FUNCTION_BLOCK FB_SlaveArm
VAR
	//
	M_TESTfLAG:BOOL:=FALSE;
	m_jnt5Planner:Cubic_Polynomial_Interpolation;
	m_initAngle,m_initVel,m_initAcc,m_initT:REAL;
	m_targetAngle,m_targetVel,m_targetAcc:REAL;
	m_cmdAngle,m_cmdVel,m_cmdAcc:REAL;
	m_initFlag:BOOL:=FALSE;
	m_finishFlag:BOOL:=TRUE;
	m_endT:REAL:=5;
	m_dT:REAL:=0.0025;
	m_T:REAL:=0;
	// arm index, from 1 to 4
	m_armIdx: INT;
	
	// joints
	m_joints :ARRAY[1..g_sJntNum] OF FB_SlaveJoint;
	
	//  panel and insturment detect
	m_panelInstrumentOnIO AT%I*	:UDINT;
	m_panelDetect :FB_PanelDetect;
	m_instruDetect :FB_InstrumentDetect;
	m_instruNearDetect :FB_InstruNearDetect;
	m_panelOnFlag :BOOL:=FALSE;
	m_instruOnFlag :BOOL:=FALSE;
	m_instruNearFlag :BOOL:=FALSE;

	
	// trocar and  adjust detect
	m_adjustIO AT%I* :UDINT;
	m_adjustDetect :FB_AdjustDetect;
	m_trocarDetect : FB_TrocarDetect;
	m_adjustOnFlag :BOOL;
	m_trocarOnFlag :BOOL :=FALSE;
	m_adjustFallEdge :BOOL:=false;
	m_adjustFallEdgeDetect : F_TRIG;
	
	//arm light out to drive
	m_lightIO AT %Q* :DINT;
	
	//endoscope type and posture switch
	m_endoscopeTypeSwitch : FB_IOToggleCheck;
	m_endoscopePostureSwitch : FB_IOToggleCheck;
	
	// instrument instance
	m_instrument : FB_Instrument;
	
	// instrument invasion depth before it's unmounted
	m_instruInvasionDepth :LREAL;

	// arm cartesian data, defined in each arm origin
	m_curCartPose	:ST_Frame;
	m_curCartTwist: Vec6d;
	m_cmdCartTwist :Vec6d;
	m_cmdCartPose:ST_Frame;
	
	// arm joint data
	m_curMotorPos :Vec8d;
	m_curLinkPos :Vec8d;
	m_curLinkSingle :Vec8d;
	m_curJntPos :Vec8d;
	m_curDHJntPos :Vec6d;
	m_curGripAngle :LREAL;
	m_curJntVel :Vec8d;
	m_curDHJntVel :Vec6d;
	m_curJntTrq :Vec8d;
	m_rawJntCurrent :Vec8d;
	m_filtJntCurrent :Vec8d;
	m_cmdJntTrq :Vec8d;
	m_cmdJntCurrent : Vec8d;
	m_cmdJntPos :Vec8d;
	m_cmdJntVel :Vec8d;
		
	// arm dynamic data
	m_jntGravity : Vec8d:=g_zeroVec8d;
	m_jntMassMat : Mat3d;
	
	// arm jacobian and inverse
	m_jaco : Mat6d;
	
	// simulated status
	m_simJntPos :Vec8d;
	m_simDHJntPos :Vec6d;
	m_simGripAngle :LREAL;
	m_simCartPose : ST_Frame;
	m_simJaco : Mat6d;
	m_simJacoInv :Mat6d;
	m_isSingularity:BOOL:=false;
	
	// joint position controller
	m_jntPIDCtrl :ARRAY[1..g_sJntNum] OF FB_PID;
	
	// rising edge generator for instrument information reading
	m_ReadLDP:R_TRIG;
	
	// code execute time measure
	m_codeTime : Profiler;

	// output arm light
	m_SdoWrite:ARRAY [1..2] OF FB_EcCoESdoWrite;
	
	//IP of operating arm
	m_armNetId:T_AmsNetId; 	
	
	//Joint port number
	m_jointAddrJ8:UINT;	
	m_jointAddrPbox:UINT;	
	m_autoLogoutTon: TON;
	g_autoLogOutTRIG: R_TRIG;
	m_logStep: INT;
	m_actualNum: INT;
	m_registerNum: INT;
	m_register: INT;
	m_accountRepeat:BOOL;
	g_targetRatedCurrent: ARRAY[1..g_sJntNum] OF LREAL := [8(800)];

	
	fbSocketConnect      :FB_SocketConnect;
	fbSocketSend         :FB_SocketSend;;;
	fbSocketReceive      :FB_SocketReceive;
	bExecute:BOOL := TRUE;
	hSocket:T_hSocket;
	arrSendData: ARRAY [0..240] OF BYTE ;
	arrReadData: ARRAY [0..240] OF BYTE ;//read
	arrRFIDData: ARRAY [0..240] OF BYTE ;
	bSend   :BOOL;
	bReceive:BOOL;
	iStepRFID: INT;
	uiRFIDReadSN: ULINT;
	iStepRFIDOnLine: INT;
	fbTonRFID: TON;
	fbTonRFIDOnLine: TON;
	fbTonRFIDOnLineStep: TON;	
	g_offLineRFID:BOOL;
	m_offLineRFID:BOOL;
	
	fbTonCLK1:TON;
	fbTonCLK2:TON;
	
	uiRFIDRead:ULINT;
	wCRCReadSum:ULINT;
	g_readedRFID:BOOL;
	fbTonReadData:TON;
	
	
	wCRC16:WORD;
	g_moveMode:INT;
	g_energyType:INT;
	uiRFIDWrite:UINT;
	g_writedRFID:BOOL;
	
	g_RFIDinstruSN:ULINT;
	
	SNMid:INT;
	g_informationVerificationPassed:BOOL;
	g_instruSN:ULINT;
	m_writeRFIDTimes:DINT;
	m_writeInstrument_pos_L1:LREAL;
	m_writeInstrument_pos_L2:LREAL;
	m_writeInstrument_pos_L3:LREAL;
	m_readRFIDTimes:DINT;
	m_readInstrument_pos_L1:LREAL;
	m_readInstrument_pos_L2:LREAL;
	m_readInstrument_pos_L3:LREAL;
	
	fbTonRFIDReaded:TON;
	stateMachineMid: E_SlaveArmState;

	g_lastInstruJntPos: Vec5d;
	fbTon: TON;
	fbTon_Logout: TON;
	startFlag:BOOL;
	m_writeSdoStart: BOOL;
	m_writeSdoTimeStart: BOOL;
	m_writeSdoFinished: BOOL;
	m_SNWritten: BOOL;
	m_SNWriteStart: BOOL;
	m_bReadRecipeStep:   INT := 1;
	m_saveAccount:BOOL;
	m_saveCaliLinkEncoder:BOOL;
	RecipeManCommands:   RecipeManCommands;
	m_writePurposeSdoStart: BOOL;
	m_getSysTime:GETSYSTEMTIME;
	m_fileTime:T_FILETIME;
	m_time:STRING;
	m_timeNow:TIMESTRUCT;
	//mes
	m_serialNumOld:STRING;
	m_curTestCyclesOld:INT;
END_VAR

PROPERTY adjustFallEdge : BOOL
GET
adjustFallEdge := m_adjustFallEdge;
END_GET
END_PROPERTY

PROPERTY adjustOn : bool
GET
adjustOn := m_adjustOnFlag;
END_GET
END_PROPERTY

PROPERTY armIdx : int
GET
armIdx:=m_armIdx;
END_GET
END_PROPERTY

METHOD PROTECTED calcJaco : BOOL
VAR_IN_OUT CONSTANT
	i_DHJntPos :Vec6d;
END_VAR
VAR_IN_OUT
	r_jaco :Mat6d;
END_VAR
VAR_INPUT
END_VAR

VAR
	d1, L, a, b :LREAL;
	q3:LREAL;

	c1,c2,c4,c5,c6,c7 :LREAL;
	s1,s2,s4,s5,s6,s7 :LREAL;

END_VAR
d1:=GVL_SlaveArmKinematic.g_d1;
L:=m_instrument.instruTypeInfo.m_rodLength;
a:=m_instrument.instruTypeInfo.m_headLength;
b:=m_instrument.instruTypeInfo.m_fingerLength;

q3:=i_DHJntPos[3];
c1:=COS(i_DHJntPos[1]);
c2:=COS(i_DHJntPos[2]);
c4:=COS(i_DHJntPos[4]);
c5:=COS(i_DHJntPos[5]);
c6:=COS(i_DHJntPos[6]);

s1:=SIN(i_DHJntPos[1]);
s2:=SIN(i_DHJntPos[2]);
s4:=SIN(i_DHJntPos[4]);
s5:=SIN(i_DHJntPos[5]);
s6:=SIN(i_DHJntPos[6]);

// jacobian with DH joints
r_jaco[1,1]:=b*(c6*(c5*(c1*s4 - c2*c4*s1) + s1*s2*s5) - s6*(c1*c4 + c2*s1*s4)) + a*(c5*(c1*s4 - c2*c4*s1) + s1*s2*s5) - L*s1*s2 + q3*s1*s2;
r_jaco[1,2]:=-c1*(a*(c2*s5 + c4*c5*s2) - L*c2 + q3*c2 + b*(c6*(c2*s5 + c4*c5*s2) + s2*s4*s6));
r_jaco[1,3]:=-c1*s2;
r_jaco[1,4]:=s1*s2*(a*(c2*s5 + c4*c5*s2) + b*(c6*(c2*s5 + c4*c5*s2) + s2*s4*s6)) - c2*(b*(c6*(c5*(c1*s4 - c2*c4*s1) + s1*s2*s5) - s6*(c1*c4 + c2*s1*s4)) + a*(c5*(c1*s4 - c2*c4*s1) + s1*s2*s5));
r_jaco[1,5]:=- (a*(c2*s5 + c4*c5*s2) + b*(c6*(c2*s5 + c4*c5*s2) + s2*s4*s6))*(c1*c4 + c2*s1*s4) - s2*s4*(b*(c6*(c5*(c1*s4 - c2*c4*s1) + s1*s2*s5) - s6*(c1*c4 + c2*s1*s4)) + a*(c5*(c1*s4 - c2*c4*s1) + s1*s2*s5));
r_jaco[1,6]:= b*(c6*(c5*(c1*s4 - c2*c4*s1) + s1*s2*s5) - s6*(c1*c4 + c2*s1*s4))*(c2*c5 - c4*s2*s5) + b*(s5*(c1*s4 - c2*c4*s1) - c5*s1*s2)*(c6*(c2*s5 + c4*c5*s2) + s2*s4*s6);


r_jaco[2,1]:=0;
r_jaco[2,2]:=c1*(a*(c5*(s1*s4 + c1*c2*c4) - c1*s2*s5) + b*(c6*(c5*(s1*s4 + c1*c2*c4) - c1*s2*s5) - s6*(c4*s1 - c1*c2*s4)) + L*c1*s2 - q3*c1*s2) - s1*(b*(c6*(c5*(c1*s4 - c2*c4*s1) + s1*s2*s5) - s6*(c1*c4 + c2*s1*s4)) + a*(c5*(c1*s4 - c2*c4*s1) + s1*s2*s5) - L*s1*s2 + q3*s1*s2);
r_jaco[2,3]:= c2;
r_jaco[2,4]:=- s1*s2*(a*(c5*(s1*s4 + c1*c2*c4) - c1*s2*s5) + b*(c6*(c5*(s1*s4 + c1*c2*c4) - c1*s2*s5) - s6*(c4*s1 - c1*c2*s4))) - c1*s2*(b*(c6*(c5*(c1*s4 - c2*c4*s1) + s1*s2*s5) - s6*(c1*c4 + c2*s1*s4)) + a*(c5*(c1*s4 - c2*c4*s1) + s1*s2*s5));
r_jaco[2,5]:=(a*(c5*(s1*s4 + c1*c2*c4) - c1*s2*s5) + b*(c6*(c5*(s1*s4 + c1*c2*c4) - c1*s2*s5) - s6*(c4*s1 - c1*c2*s4)))*(c1*c4 + c2*s1*s4) - (b*(c6*(c5*(c1*s4 - c2*c4*s1) + s1*s2*s5) - s6*(c1*c4 + c2*s1*s4)) + a*(c5*(c1*s4 - c2*c4*s1) + s1*s2*s5))*(c4*s1 - c1*c2*s4);
r_jaco[2,6]:=b*(c6*(c5*(c1*s4 - c2*c4*s1) + s1*s2*s5) - s6*(c1*c4 + c2*s1*s4))*(s5*(s1*s4 + c1*c2*c4) + c1*c5*s2) - b*(s5*(c1*s4 - c2*c4*s1) - c5*s1*s2)*(c6*(c5*(s1*s4 + c1*c2*c4) - c1*s2*s5) - s6*(c4*s1 - c1*c2*s4));

r_jaco[3,1]:=a*(c5*(s1*s4 + c1*c2*c4) - c1*s2*s5) + b*(c6*(c5*(s1*s4 + c1*c2*c4) - c1*s2*s5) - s6*(c4*s1 - c1*c2*s4)) + L*c1*s2 - q3*c1*s2;
r_jaco[3,2]:=-s1*(a*(c2*s5 + c4*c5*s2) - L*c2 + q3*c2 + b*(c6*(c2*s5 + c4*c5*s2) + s2*s4*s6));
r_jaco[3,3]:=-s1*s2;
r_jaco[3,4]:=- c2*(a*(c5*(s1*s4 + c1*c2*c4) - c1*s2*s5) + b*(c6*(c5*(s1*s4 + c1*c2*c4) - c1*s2*s5) - s6*(c4*s1 - c1*c2*s4))) - c1*s2*(a*(c2*s5 + c4*c5*s2) + b*(c6*(c2*s5 + c4*c5*s2) + s2*s4*s6));
r_jaco[3,5]:=- (a*(c2*s5 + c4*c5*s2) + b*(c6*(c2*s5 + c4*c5*s2) + s2*s4*s6))*(c4*s1 - c1*c2*s4) - s2*s4*(a*(c5*(s1*s4 + c1*c2*c4) - c1*s2*s5) + b*(c6*(c5*(s1*s4 + c1*c2*c4) - c1*s2*s5) - s6*(c4*s1 - c1*c2*s4)));
r_jaco[3,6]:=b*(c6*(c5*(s1*s4 + c1*c2*c4) - c1*s2*s5) - s6*(c4*s1 - c1*c2*s4))*(c2*c5 - c4*s2*s5) + b*(c6*(c2*s5 + c4*c5*s2) + s2*s4*s6)*(s5*(s1*s4 + c1*c2*c4) + c1*c5*s2);

r_jaco[4,1]:=0;
r_jaco[4,2]:=-s1;
r_jaco[4,3]:=0;
r_jaco[4,4]:=-c1*s2;
r_jaco[4,5]:=c1*c2*s4 - c4*s1;
r_jaco[4,6]:=s5*(s1*s4 + c1*c2*c4) + c1*c5*s2;

r_jaco[5,1]:=-1;
r_jaco[5,2]:=0;
r_jaco[5,3]:=0;
r_jaco[5,4]:=c2;
r_jaco[5,5]:=s2*s4;
r_jaco[5,6]:=c4*s2*s5 - c2*c5;

r_jaco[6,1]:=0;
r_jaco[6,2]:=c1;
r_jaco[6,3]:=0;
r_jaco[6,4]:=-s1*s2;
r_jaco[6,5]:=c1*c4 + c2*s1*s4;
r_jaco[6,6]:=c5*s1*s2 - s5*(c1*s4 - c2*c4*s1);
END_METHOD

METHOD PROTECTED checkIO : BOOL

VAR

	i: INT;
	ReturnDwordRead:DWORD;
	ReturnDwordWrite:DWORD;
END_VAR
// check adjust button
m_adjustOnFlag := m_adjustDetect.run(m_adjustIO);
m_adjustFallEdgeDetect(CLK:=m_adjustOnFlag, Q=>m_adjustFallEdge);

// check trocar
m_trocarOnFlag := m_trocarDetect.run(m_adjustIO);

// check panel and instrument
m_panelOnFlag := m_panelDetect.run(m_panelInstrumentOnIO);
m_instruOnFlag :=m_instruDetect.run(m_panelInstrumentOnIO);
m_instruNearFlag := m_instruNearDetect.run(m_panelInstrumentOnIO);

//read instrument information
IF FALSE = m_instruOnFlag THEN
	m_instrument.reset();
END_IF


m_ReadLDP(CLK:= m_instruOnFlag, Q=>startFlag );
// try to read again if instrument ID is undefined
startFlag := startFlag OR m_instrument.onChipData.m_ErrorID = 1 OR GVL_InstruTestUIVars.g_readInstruinformation;
m_instrument.readParameters(startFlag);

GVL_InstruTestUIVars.g_readInstruinformationFlag:=m_instrument.onChipData.m_InstruReadSucceed;
// check endoscope type and posture 
IF m_endoscopeTypeSwitch.check((m_panelInstrumentOnIO AND 16#20)=32) THEN
	IF m_instrument.curScopeType = EndoScopeType_30 THEN
		m_instrument.nextScopeType := EndoscopeType_0;
	ELSE
		m_instrument.nextScopeType := EndoscopeType_30;
	END_IF
END_IF
IF m_endoscopePostureSwitch.check((m_panelInstrumentOnIO AND 16#10)=16) AND m_instrument.curScopeType = EndoScopeType_30  THEN
	IF m_instrument.curScopePosture = EndoScopePosture_HeadDown THEN
		m_instrument.nextScopePosture := EndoscopePosture_HeadUp;
	ELSE
		m_instrument.nextScopePosture := EndoScopePosture_HeadDown;
	END_IF
END_IF

IF GVL_InstruTestUIVars.g_incInstruNumOfUses THEN
	GVL_InstruTestUIVars.g_jnt5RotateFlag:=TRUE;
	m_writeSdoTimeStart := TRUE;
ELSE
	IF m_writeSdoTimeStart THEN
		IF   NOT m_writeSdoFinished THEN
			m_writeSdoFinished :=instrument.addNumOfUseToChip();

		ELSE
			m_writeSdoTimeStart :=FALSE;
			m_writeSdoFinished:=FALSE;
		END_IF
	END_IF
END_IF

IF GVL_InstruTestUIVars.g_clearInstruNumOfUses THEN
	m_writeSdoStart := TRUE;
ELSE
	IF m_writeSdoStart THEN
		IF   NOT m_writeSdoFinished THEN
			m_writeSdoFinished :=instrument.clearNumOfUseToChip();

		ELSE
			m_writeSdoStart :=FALSE;
			m_writeSdoFinished:=FALSE;
		END_IF
	END_IF
END_IF

// write SN to CoE
IF GVL_InstruTestUIVars.g_writeSNFlag THEN
	m_SNWriteStart := TRUE;
ELSE
	IF m_SNWriteStart THEN
		IF   NOT m_SNWritten THEN
			m_SNWritten := instrument.writeSNToChip(STRING_TO_ULINT(GVL_InstruTestUIVars.g_newInstruSN));
		ELSE
			m_SNWriteStart :=FALSE;
			m_SNWritten:=FALSE;
		END_IF
	END_IF
END_IF

IF GVL_InstruTestUIVars.g_writeInstruPurpose AND m_instrument.onChipData.m_InstruReadSucceed THEN
	m_writePurposeSdoStart := TRUE;
ELSE
	IF m_writePurposeSdoStart THEN
		IF   NOT m_writeSdoFinished THEN
			m_writeSdoFinished :=instrument.writePurpose();

		ELSE
			m_writePurposeSdoStart :=FALSE;
			m_writeSdoFinished:=FALSE;
		END_IF
	END_IF
END_IF

GVL_InstruTestUIVars.g_maxAngle:=INT_TO_REAL(REAL_TO_INT(m_instrument.instruTypeInfo.m_maxGripAngle/g_deg2Rad));
GVL_InstruTestUIVars.g_maxRoll:=INT_TO_REAL(REAL_TO_INT(m_instrument.instruTypeInfo.m_rollLimit/g_deg2Rad));
GVL_InstruTestUIVars.g_maxPitch:=INT_TO_REAL(REAL_TO_INT(m_instrument.instruTypeInfo.m_pitchLimit/g_deg2Rad));
GVL_InstruTestUIVars.g_maxYaw:=INT_TO_REAL(REAL_TO_INT(m_instrument.instruTypeInfo.m_yawLimit/g_deg2Rad));
GVL_InstruTestUIVars.g_maxAngleEnable:=GVL_InstruTestUIVars.g_targetGripAng*g_deg2rad>m_instrument.instruTypeInfo.m_maxGripAngle;
GVL_InstruTestUIVars.g_maxRollEnable:=ABS(GVL_InstruTestUIVars.g_targetRollAng)*g_deg2rad>m_instrument.instruTypeInfo.m_rollLimit;
GVL_InstruTestUIVars.g_maxPitchEnable:=ABS(GVL_InstruTestUIVars.g_targetPitchAng)*g_deg2rad>m_instrument.instruTypeInfo.m_pitchLimit;
GVL_InstruTestUIVars.g_maxYawEnable:=ABS(GVL_InstruTestUIVars.g_targetYawAng)*g_deg2rad>m_instrument.instruTypeInfo.m_yawLimit;

GVL_InstruTestUIVars.g_incInstruNumOfUses:=FALSE;
GVL_InstruTestUIVars.g_clearInstruNumOfUses:=FALSE;
GVL_InstruTestUIVars.g_writeSNFlag:=FALSE;
GVL_InstruTestUIVars.g_writeInstruPurpose:=FALSE;

GVL_InstruTestUIVars.g_instruNumberOfUses:=ULINT_TO_UINT( m_instrument.onChipData.m_InstruusageCounts);
GVL_InstruTestUIVars.g_instruNumberOfAllUses:=ULINT_TO_UINT( m_instrument.onChipData.m_InstruUsageCounts);
GVL_InstruTestUIVars.g_readInstruPurpose:=ULINT_TO_UINT( m_instrument.onChipData.m_InstruPurpose);
GVL_InstruTestUIVars.g_readPurposeTime:=ULINT_TO_UINT( m_instrument.onChipData.m_InstruPurposeTime);

GVL_InstruTestUIVars.g_instruSN:=ULINT_TO_STRING(m_instrument.onChipData.m_InstruseriesNum);
IF (LEN(GVL_InstruTestUIVars.g_instruSN)=10)THEN
	GVL_InstruTestUIVars.g_instruSN:=concat('00',GVL_InstruTestUIVars.g_instruSN);
ELSIF  (LEN(GVL_InstruTestUIVars.g_instruSN)=11)THEN
	GVL_InstruTestUIVars.g_instruSN:=concat('0',GVL_InstruTestUIVars.g_instruSN);
ELSE
	GVL_InstruTestUIVars.g_instruSN:=GVL_InstruTestUIVars.g_instruSN;
END_IF

GVL_InstruTestUIVars.g_rotationActualCurrent:=m_filtJntCurrent[7];
GVL_InstruTestUIVars.g_pitchActualCurrent:=m_filtJntCurrent[6];
GVL_InstruTestUIVars.g_deviationActualCurrent:=m_filtJntCurrent[4];
//***************************修改电流极限**************************//
GVL_InstruTestUIVars.g_actualRatedCurrent:=g_targetRatedCurrent;
IF GVL_InstruTestUIVars.g_modifyRatedCurrent THEN
	GVL_InstruTestUIVars.g_modifyRatedCurrent:=FALSE;
	FOR i:=1 TO 8 BY 1 DO 
		GVL_InstruTestUIVars.g_actualRatedCurrent[i]:=GVL_InstruTestUIVars.g_targetRatedCurrent;
		g_targetRatedCurrent[i]:=GVL_InstruTestUIVars.g_targetRatedCurrent;
	END_FOR
END_IF
IF GVL_InstruTestUIVars.g_rotationTargetCurrent=0 THEN GVL_InstruTestUIVars.g_rotationTargetCurrent:=100; END_IF
IF GVL_InstruTestUIVars.g_pitchTargetCurrent=0 THEN GVL_InstruTestUIVars.g_pitchTargetCurrent:=100; END_IF
IF GVL_InstruTestUIVars.g_deviationTargetCurrent=0 THEN GVL_InstruTestUIVars.g_deviationTargetCurrent:=100; END_IF
IF GVL_InstruTestUIVars.g_deviationTargetCurrent=0 THEN GVL_InstruTestUIVars.g_deviationTargetCurrent:=100; END_IF
IF GVL_InstruTestUIVars.g_account.actualPermission=2 AND GVL_InstruTestUIVars.g_stateMachine=SlaveArmState_InstruManualTest  THEN
	GVL_InstruTestUIVars.g_actualRatedCurrent[7]:=GVL_InstruTestUIVars.g_rotationTargetCurrent;
	GVL_InstruTestUIVars.g_actualRatedCurrent[6]:=GVL_InstruTestUIVars.g_pitchTargetCurrent;
	GVL_InstruTestUIVars.g_actualRatedCurrent[5]:=GVL_InstruTestUIVars.g_deviationTargetCurrent;
	GVL_InstruTestUIVars.g_actualRatedCurrent[4]:=GVL_InstruTestUIVars.g_deviationTargetCurrent;
END_IF
IF GVL_InstruTestUIVars.g_stateMachine=SlaveArmState_InstruAutoTest AND GVL_MES.g_autoTestMode=3 THEN
	GVL_InstruTestUIVars.g_actualRatedCurrent[4]:=540;
	GVL_InstruTestUIVars.g_actualRatedCurrent[5]:=540;
	GVL_InstruTestUIVars.g_actualRatedCurrent[6]:=540;
	GVL_InstruTestUIVars.g_actualRatedCurrent[7]:=540;
	IF m_instrument.onChipData.m_InstruReadSucceed AND(InstruType_CauteryHook=m_instrument.m_instruType OR InstruType_CauterySpatula=m_instrument.m_instruType) THEN
	GVL_InstruTestUIVars.g_actualRatedCurrent[4]:=270;
	GVL_InstruTestUIVars.g_actualRatedCurrent[5]:=270;
	GVL_InstruTestUIVars.g_actualRatedCurrent[6]:=270;
	GVL_InstruTestUIVars.g_actualRatedCurrent[7]:=270;
	END_IF
END_IF
//Account
GVL_InstruTestUIVars.g_account.memoryAccountNumber[0] :='admin';
GVL_InstruTestUIVars.g_account.memoryPassWord[0] :='yfAGIBOT2025';
GVL_InstruTestUIVars.g_account.memoryPermission[0] :=1;
GVL_InstruTestUIVars.g_account.memoryName[0] :='admin';
GVL_InstruTestUIVars.g_account.memoryWorkNum[0] :=101;
GVL_InstruTestUIVars.g_account.memoryDisable[0]:=FALSE;
CASE m_logStep OF 
	0: 
	  IF GVL_InstruTestUIVars.g_account.logOn THEN 
		   m_logStep:=5;
		   m_actualNum:=-1;
		  GVL_InstruTestUIVars.g_account.logOn:=FALSE;
	  END_IF
	5:
	FOR i:= 0 TO 50 BY 1 DO
		IF GVL_InstruTestUIVars.g_account.actualAccountNumber = GVL_InstruTestUIVars.g_account.memoryAccountNumber[i] AND GVL_InstruTestUIVars.g_account.actualAccountNumber <> ''THEN
			m_actualNum:=i;
			m_logStep:=10;
		ELSE
			IF m_actualNum=-1 THEN
				GVL_InstruTestUIVars.g_account.prompt:='Account Err';
				m_logStep:=0;
			END_IF
		END_IF
	END_FOR
	10:
	IF GVL_InstruTestUIVars.g_account.actualPassWord = GVL_InstruTestUIVars.g_account.memoryPassWord[m_actualNum] AND GVL_InstruTestUIVars.g_account.actualAccountNumber <> ''THEN
		m_logStep:=12;
	ELSE
		GVL_InstruTestUIVars.g_account.prompt:='PassWord Err';
		m_logStep:=0;
	END_IF
	12:
	IF GVL_InstruTestUIVars.g_account.memoryDisable[m_actualNum] THEN
		GVL_InstruTestUIVars.g_account.prompt:='No Enable';
		m_logStep:=0;
	ELSE
		m_logStep:=15;
	END_IF
	15:
	GVL_InstruTestUIVars.g_account.actualPermission := GVL_InstruTestUIVars.g_account.memoryPermission[m_actualNum];
	GVL_InstruTestUIVars.g_account.actualWorkNum := GVL_InstruTestUIVars.g_account.memoryWorkNum[m_actualNum];
	GVL_InstruTestUIVars.g_account.actualName := GVL_InstruTestUIVars.g_account.memoryName[m_actualNum];
	GVL_InstruTestUIVars.g_account.autoLogOut:=FALSE;
	GVL_InstruTestUIVars.g_account.prompt:='Login Succeeded';
	m_logStep:=0;
END_CASE

FOR i:=1 TO 5 DO 
	IF stateMachineMid<>GVL_InstruTestUIVars.g_stateMachine OR ABS(GVL_InstruTestUIVars.g_curInstruJntPos[i]-g_lastInstruJntPos[i])>0.01 THEN
		GVL_InstruTestUIVars.g_account.autoLogOut:=FALSE;
	ELSE
		IF NOT GVL_InstruTestUIVars.g_account.autoLogOut THEN 
			IF fbTon_Logout.Q THEN
				GVL_InstruTestUIVars.g_account.autoLogOut:=TRUE;
			END_IF
		END_IF
	END_IF
END_FOR
	fbTon(IN:= NOT fbTon.Q, PT:=T#10MS );
	IF fbTon.Q THEN
		g_lastInstruJntPos:= GVL_InstruTestUIVars.g_curInstruJntPos;
	END_IF
stateMachineMid:=GVL_InstruTestUIVars.g_stateMachine;
fbTon_Logout(IN:=NOT GVL_InstruTestUIVars.g_account.autoLogOut,PT:=T#0.1S);


m_autoLogoutTon(IN:=GVL_InstruTestUIVars.g_account.autoLogOut,PT:=T#1H);
g_autoLogOutTRIG(CLK:=m_autoLogoutTon.Q);
IF GVL_InstruTestUIVars.g_account.logOut OR g_autoLogOutTRIG.Q THEN
	GVL_InstruTestUIVars.g_account.actualPermission :=0;
	GVL_InstruTestUIVars.g_account.actualAccountNumber :='';
	GVL_InstruTestUIVars.g_account.actualPassWord :='';
	GVL_InstruTestUIVars.g_account.actualWorkNum :=0;
	GVL_InstruTestUIVars.g_account.actualName :='';
	GVL_InstruTestUIVars.g_account.logOut:=FALSE;
	GVL_InstruTestUIVars.g_account.prompt:='';
END_IF
IF GVL_InstruTestUIVars.g_clearInformation THEN
	GVL_InstruTestUIVars.g_account.actualAccountNumber :='';
	GVL_InstruTestUIVars.g_account.actualPassWord :='';
	GVL_InstruTestUIVars.g_account.actualWorkNum :=0;
	GVL_InstruTestUIVars.g_account.actualName :='';
	GVL_InstruTestUIVars.g_account.prompt:='';
	GVL_InstruTestUIVars.g_account.registerAccountNumber :='';
	GVL_InstruTestUIVars.g_account.registerPassWord :='';
	GVL_InstruTestUIVars.g_account.registerWorkNum :=0;
	GVL_InstruTestUIVars.g_account.registerName :='';
	GVL_InstruTestUIVars.g_account.prompt:='';
	GVL_InstruTestUIVars.g_clearInformation:=FALSE;
END_IF
IF GVL_InstruTestUIVars.g_account.registerPermission<>2 AND GVL_InstruTestUIVars.g_account.registerPermission<>3 AND
	GVL_InstruTestUIVars.g_account.registerPermission<>4 THEN
//	GVL_InstruTestUIVars.g_account.registerPermission:=4;
END_IF
m_getSysTime(timeLoDW=>m_fileTime.dwLowDateTime, timeHiDW=>m_fileTime.dwHighDateTime);
m_timeNow:=FILETIME_TO_SYSTEMTIME(m_fileTime);
m_timeNow.wHour:=m_timeNow.wHour+8;
IF m_timeNow.wHour>23 THEN
	m_timeNow.wHour:=m_timeNow.wHour-24;
END_IF
m_time:=SYSTEMTIME_TO_STRING(m_timeNow);
CASE m_registerNum OF 
	0:
	  IF GVL_InstruTestUIVars.g_account.register THEN 
		  GVL_InstruTestUIVars.g_account.register:=FALSE;
		  GVL_InstruTestUIVars.g_account.prompt:='';
		  m_accountRepeat:=FALSE;
		  m_register:=-1;
		  m_registerNum:=5;
	  END_IF
	5:
	FOR i:= 0 TO 50 BY 1 DO
      IF  GVL_InstruTestUIVars.g_account.registerAccountNumber <> GVL_InstruTestUIVars.g_account.memoryAccountNumber[i] AND GVL_InstruTestUIVars.g_account.registerAccountNumber <> ''THEN
		;	  
	  ELSE
		  m_accountRepeat:=TRUE;
	  END_IF
	END_FOR
	m_registerNum:=6;
	6:
	IF m_accountRepeat THEN
		GVL_InstruTestUIVars.g_account.prompt:='Account Repeat';
		m_registerNum:=0;
	ELSE
		m_registerNum:=10;
	END_IF
	10:
	IF GVL_InstruTestUIVars.g_account.registerPassWord<> '' THEN
		m_registerNum:=15;
	ELSE
		GVL_InstruTestUIVars.g_account.prompt:='No PassWord';
		m_registerNum:=0;
	END_IF
	15:
	IF GVL_InstruTestUIVars.g_account.registerWorkNum<> 0 THEN
		m_registerNum:=20;
	ELSE
		GVL_InstruTestUIVars.g_account.prompt:='No WorkNum';
		m_registerNum:=0;
	END_IF
	20:
	IF GVL_InstruTestUIVars.g_account.registerName<> '' THEN
		m_registerNum:=25;
	ELSE
		GVL_InstruTestUIVars.g_account.prompt:='No Name';
		m_registerNum:=0;
	END_IF
	25:
	IF GVL_InstruTestUIVars.g_account.registerPermission<> 0 THEN
		m_registerNum:=30;
	ELSE
		GVL_InstruTestUIVars.g_account.prompt:='No Permission';
		m_registerNum:=0;
	END_IF
	30:
	FOR i:= 50 TO 0 BY -1 DO
      IF  '' = GVL_InstruTestUIVars.g_account.memoryAccountNumber[i] THEN
		 m_register:=i;
		 m_registerNum:=35;
	  ELSE
		  IF m_register=-1 THEN
			 GVL_InstruTestUIVars.g_account.prompt:='No Room';
			 m_registerNum:=0;	
		END_IF
	  END_IF
 	END_FOR
	35:
	GVL_InstruTestUIVars.g_account.memoryAccountNumber[m_register]:=GVL_InstruTestUIVars.g_account.registerAccountNumber;
	GVL_InstruTestUIVars.g_account.memoryPassWord[m_register]:=GVL_InstruTestUIVars.g_account.registerPassWord;
	GVL_InstruTestUIVars.g_account.memoryWorkNum[m_register]:=GVL_InstruTestUIVars.g_account.registerWorkNum;
	GVL_InstruTestUIVars.g_account.memoryName[m_register]:=GVL_InstruTestUIVars.g_account.registerName;
	GVL_InstruTestUIVars.g_account.memoryPermission[m_register]:=GVL_InstruTestUIVars.g_account.registerPermission;
	IF GVL_InstruTestUIVars.g_account.registerPermission=1 THEN
		GVL_InstruTestUIVars.g_account.memoryPermission[m_register]:=4;
	END_IF
	GVL_InstruTestUIVars.g_account.memoryTime[m_register]:=m_time;
	GVL_InstruTestUIVars.g_account.prompt:='Register Succeeded';
	m_registerNum:=0;
	m_saveAccount:=TRUE;
END_CASE

GVL_InstruTestUIVars.g_accountSN := LIMIT(1,GVL_InstruTestUIVars.g_accountSN, 50);
IF GVL_InstruTestUIVars.g_accountDelete THEN 
	GVL_InstruTestUIVars.g_accountDelete:=FALSE;
	m_saveAccount:=TRUE;
	GVL_InstruTestUIVars.g_account.memoryAccountNumber[GVL_InstruTestUIVars.g_accountSN]:='';
	GVL_InstruTestUIVars.g_account.memoryPassWord[GVL_InstruTestUIVars.g_accountSN]:='';
	GVL_InstruTestUIVars.g_account.memoryWorkNum[GVL_InstruTestUIVars.g_accountSN]:=0;
	GVL_InstruTestUIVars.g_account.memoryName[GVL_InstruTestUIVars.g_accountSN]:='';
	GVL_InstruTestUIVars.g_account.memoryPermission[GVL_InstruTestUIVars.g_accountSN]:=0;
	GVL_InstruTestUIVars.g_account.memoryTime[GVL_InstruTestUIVars.g_accountSN]:='';
END_IF
IF GVL_InstruTestUIVars.g_disableAccount THEN 
	GVL_InstruTestUIVars.g_disableAccount:=FALSE;
	IF GVL_InstruTestUIVars.g_account.memoryDisable[GVL_InstruTestUIVars.g_accountSN] THEN
		GVL_InstruTestUIVars.g_account.memoryDisable[GVL_InstruTestUIVars.g_accountSN]:=FALSE;
	ELSE
		GVL_InstruTestUIVars.g_account.memoryDisable[GVL_InstruTestUIVars.g_accountSN]:=TRUE;
	END_IF
END_IF	
FOR i:=1 TO 50 BY 1 DO 
	IF GVL_InstruTestUIVars.g_account.memoryAccountNumber[i]='' THEN
		GVL_InstruTestUIVars.g_account.memoryDisable[i]:=FALSE;
	END_IF
END_FOR
GVL_InstruTestUIVars.g_queryAccountSN := LIMIT(0,GVL_InstruTestUIVars.g_queryAccountSN, 50);
IF GVL_InstruTestUIVars.g_queryAccountFlag THEN 
	GVL_InstruTestUIVars.g_queryAccountFlag:=FALSE;
	GVL_InstruTestUIVars.g_queryAccountNumber:='';
	GVL_InstruTestUIVars.g_queryPassWord:='';
	GVL_InstruTestUIVars.g_queryPermission:=0;
	GVL_InstruTestUIVars.g_queryWorkNum:=0;
	GVL_InstruTestUIVars.g_queryName:='';
	GVL_InstruTestUIVars.g_queryTime:='';
	GVL_InstruTestUIVars.g_queryAccountNumber:=GVL_InstruTestUIVars.g_account.memoryAccountNumber[GVL_InstruTestUIVars.g_queryAccountSN];
	GVL_InstruTestUIVars.g_queryPassWord:=GVL_InstruTestUIVars.g_account.memoryPassWord[GVL_InstruTestUIVars.g_queryAccountSN];
	GVL_InstruTestUIVars.g_queryPermission:=GVL_InstruTestUIVars.g_account.memoryPermission[GVL_InstruTestUIVars.g_queryAccountSN];
	GVL_InstruTestUIVars.g_queryWorkNum:=GVL_InstruTestUIVars.g_account.memoryWorkNum[GVL_InstruTestUIVars.g_queryAccountSN];
	GVL_InstruTestUIVars.g_queryName:=GVL_InstruTestUIVars.g_account.memoryName[GVL_InstruTestUIVars.g_queryAccountSN];
	GVL_InstruTestUIVars.g_queryTime:=GVL_InstruTestUIVars.g_account.memoryTime[GVL_InstruTestUIVars.g_queryAccountSN];
END_IF
IF GVL_InstruTestUIVars.g_queryClear THEN 
	GVL_InstruTestUIVars.g_queryClear:=FALSE;
	GVL_InstruTestUIVars.g_queryAccountNumber:='';
	GVL_InstruTestUIVars.g_queryPassWord:='';
	GVL_InstruTestUIVars.g_queryPermission:=0;
	GVL_InstruTestUIVars.g_queryWorkNum:=0;
	GVL_InstruTestUIVars.g_queryName:='';
	GVL_InstruTestUIVars.g_queryTime:='';
END_IF

bExecute:=NOT fbSocketConnect.bError OR fbTon.Q;

fbSocketConnect(
	sSrvNetId:= , 
	sRemoteHost:='192.168.1.202' , 
	nRemotePort:= 4196, 
	bExecute:= bExecute, 
	tTimeout:=T#3S , 
	bBusy=> , 
	bError=> , 
	nErrId=> , 
	hSocket=>hSocket );
	
	fbSocketSend(
	sSrvNetId:= , 
	hSocket:= hSocket, 
	cbLen:= SIZEOF(arrSendData), 
	pSrc:= ADR(arrSendData), 
	bExecute:= bSend, 
	tTimeout:= T#3S, 
	bBusy=> , 
	bError=> , 
	nErrId=> );
	
	
	fbSocketReceive(
	sSrvNetId:= , 
	hSocket:=hSocket , 
	cbLen:= SIZEOF(arrReadData), 
	pDest:= ADR(arrReadData), 
	bExecute:= bReceive, 
	tTimeout:= T#3S, 
	bBusy=> , 
	bError=> , 
	nErrId=> , 
	nRecBytes=> );
	
	bSend:=FALSE;
	fbTonCLK1(IN:=NOT fbTonCLK2.Q,PT:=T#1S);
	fbTonCLK2(IN:=fbTonCLK1.Q,PT:=T#1S);
	bReceive:=fbTonCLK1.Q;
//RFID
m_instrument.readParametersRFID(GVL_InstruTestUIVars.g_readRFID);
GVL_InstruTestUIVars.g_readRFID:=FALSE;
g_informationVerificationPassed:=FALSE;
IF m_instrument.onChipData.m_InstruReadSucceedRFID AND m_instrument.onChipData.m_InstruseriesNumRFID=m_instrument.onChipData.m_InstruseriesNum  AND 
	ABS(m_instrument.onChipData.m_InstruPosRFID[1]-m_instrument.onChipData.m_InstruPos[1])<0.01 AND
	ABS(m_instrument.onChipData.m_InstruPosRFID[2]-m_instrument.onChipData.m_InstruPos[2])<0.01 AND
	ABS(m_instrument.onChipData.m_InstruPosRFID[3]-m_instrument.onChipData.m_InstruPos[3])<0.01 THEN
	
	g_informationVerificationPassed:=TRUE;
END_IF;
GVL_InstruTestUIVars.g_RFID_SN:=ULINT_TO_STRING(m_instrument.onChipData.m_InstruseriesNumRFID);
IF (LEN(GVL_InstruTestUIVars.g_RFID_SN)=10)THEN
	GVL_InstruTestUIVars.g_RFID_SN:=concat('00',GVL_InstruTestUIVars.g_RFID_SN);
ELSIF  (LEN(GVL_InstruTestUIVars.g_RFID_SN)=11)THEN
	GVL_InstruTestUIVars.g_RFID_SN:=concat('0',GVL_InstruTestUIVars.g_RFID_SN);
ELSE
	GVL_InstruTestUIVars.g_RFID_SN:=GVL_InstruTestUIVars.g_RFID_SN;
END_IF
GVL_InstruTestUIVars.m_RFIDTimes:=ULINT_TO_DINT(m_instrument.onChipData.m_InstruUsageCountsRFID);
GVL_InstruTestUIVars.m_Instrument_pos_L1:=m_instrument.onChipData.m_InstruPosRFID[1];
GVL_InstruTestUIVars.m_Instrument_pos_L2:=m_instrument.onChipData.m_InstruPosRFID[2];
GVL_InstruTestUIVars.m_Instrument_pos_L3:=m_instrument.onChipData.m_InstruPosRFID[3];
GVL_InstruTestUIVars.g_informationVerificationPassed:=g_informationVerificationPassed;
GVL_InstruTestUIVars.g_readedRFID:=m_instrument.onChipData.m_InstruReadSucceedRFID;
IF GVL_InstruTestUIVars.g_readRFID AND iStepRFID=0 THEN
	GVL_InstruTestUIVars.g_readRFID:=FALSE;
	g_readedRFID:=FALSE;
	GVL_InstruTestUIVars.g_readRFIDFlag:=FALSE;
	uiRFIDReadSN:=0;
	iStepRFID:=3;
	iStepRFIDOnLine:=0;
END_IF
IF GVL_InstruTestUIVars.g_writeRFID AND iStepRFID=0 THEN
	GVL_InstruTestUIVars.g_writeRFID:=FALSE;
	iStepRFID:=53;
	iStepRFIDOnLine:=0;
END_IF

fbTonRFID(IN:=iStepRFID=10 OR iStepRFID=60, PT:=T#5S , Q=> , ET=> );
fbTonRFIDOnLine(IN:=m_offLineRFID , PT:=T#2S , Q=> , ET=> );
fbTonRFIDOnLineStep(IN:=iStepRFIDOnLine=10 , PT:=T#1S , Q=> , ET=> );
fbTonReadData(IN:=iStepRFID=15 OR iStepRFID=65 , PT:=T#0.5S , Q=> , ET=> );
IF fbTonRFIDOnLine.Q THEN
    g_offLineRFID:=FALSE;;
END_IF

CASE iStepRFID OF
	0:
(*		CASE iStepRFIDOnLine OF   //On  Off line
			0:
			  arrReadData:=arrRFIDData;
			  arrSendData:=arrRFIDData;
			  iStepRFIDOnLine:=5;
			5:   
			  arrSendData[1]:=16#FF;
			  arrSendData[2]:=16#08;  arrSendData[3]:=16#11;
			  arrSendData[4]:=16#00;  arrSendData[5]:=16#01;
			  arrSendData[6]:=16#00;  arrSendData[7]:=16#00;
			  arrSendData[8]:=16#01;  arrSendData[9]:=16#EF;
			  arrSendData[10]:=16#7F;  arrSendData[11]:=16#32;
			  bSend:=TRUE; 
			  iStepRFIDOnLine:=10;
			10:
			  IF arrReadData[0]<>0  THEN
				  g_offLineRFID:=TRUE;
				  m_offLineRFID:=FALSE;
			  ELSE
                  m_offLineRFID:=TRUE;
			  END_IF
			  IF fbTonRFIDOnLineStep.Q THEN
			  	  iStepRFIDOnLine:=0;
			  END_IF
		END_CASE
		
	*)	
    3:                           //Read
	  arrReadData:=arrRFIDData;
	  arrSendData:=arrRFIDData;
	  iStepRFID:=5;
	5:
	  arrSendData[0]:=16#FF;
	  arrSendData[1]:=16#08;  arrSendData[2]:=16#11;
	  arrSendData[3]:=16#00;  arrSendData[4]:=16#01;
	  arrSendData[5]:=16#00;  arrSendData[6]:=16#00;
	  arrSendData[7]:=16#01;  arrSendData[8]:=16#6E;
	  arrSendData[9]:=16#1F;  arrSendData[10]:=16#F2;
	  arrSendData[11]:=16#00; 
	  bSend:=TRUE; 
	  iStepRFID:=10;
	10:
	   IF arrReadData[0]<>0  THEN
		   iStepRFID:=15;
	   END_IF
	   IF fbTonRFID.Q THEN
		   iStepRFID:=0;
	       iStepRFIDOnLine:=0;
	   END_IF
	15: 
	IF fbTonReadData.Q THEN
//	   IF arrReadData[5]=0 THEN
	   	   iStepRFID:=20;
//	   END_IF
//	   IF arrReadData[5]<>0THEN
//	   	   iStepRFID:=30;
//	   END_IF
	END_IF
    20:
	   uiRFIDRead:=0;
	   FOR i:=8 TO 108 BY 1 DO
		    uiRFIDRead:=BYTE_TO_UINT(arrReadData[i])+uiRFIDRead;
	   END_FOR
  	   iStepRFID:=25;
	 25:
//	   AryByteTo(In:=arrReadData[111] , Size:= 2, Order:=_eBYTE_ORDER._HIGH_LOW , OutVal:=wCRCReadSum );
	   wCRCReadSum:=SHL(BYTE_TO_ULINT(arrReadData[109]),8)OR BYTE_TO_ULINT(arrReadData[110]);
	   IF wCRCReadSum=uiRFIDRead THEN
	    	g_readedRFID:=TRUE;
			GVL_InstruTestUIVars.g_readRFIDFlag:=TRUE;
			uiRFIDReadSN:=0;
	   FOR i:=1 TO 8 BY 1 DO
		  uiRFIDReadSN:=SHL(BYTE_TO_ULINT(arrReadData[58+i]),64-i*8)+uiRFIDReadSN;
	  END_FOR
	  m_readRFIDTimes:=0;
	   FOR i:=1 TO 4 BY 1 DO
		  m_readRFIDTimes:=SHL(BYTE_TO_DINT(arrReadData[68+i]),32-i*8)+m_readRFIDTimes;
	  END_FOR
	  m_readInstrument_pos_L1:=0;
	  m_readInstrument_pos_L2:=0;
	  m_readInstrument_pos_L3:=0;
	   FOR i:=1 TO 4 BY 1 DO
		  m_readInstrument_pos_L1:=DINT_TO_LREAL(SHL(BYTE_TO_DINT(arrReadData[28+i]),32-i*8))/1000+m_readInstrument_pos_L1;
	  END_FOR
	   FOR i:=1 TO 4 BY 1 DO
		  m_readInstrument_pos_L2:=DINT_TO_LREAL(SHL(BYTE_TO_DINT(arrReadData[38+i]),32-i*8))/1000+m_readInstrument_pos_L2;
	  END_FOR
	   FOR i:=1 TO 4 BY 1 DO
		  m_readInstrument_pos_L3:=DINT_TO_LREAL(SHL(BYTE_TO_DINT(arrReadData[48+i]),32-i*8))/1000+m_readInstrument_pos_L3;
	  END_FOR
	  
//			AryByteTo(In:=arrReadData[61] , Size:= 12, Order:=_eBYTE_ORDER._HIGH_LOW , OutVal:=uiRFIDReadSN );
//			m_instruPurpose:=BYTE_TO_INT(arrReadData[74]);
//			AryByteTo(In:=arrReadData[47] , Size:= 2, Order:=_eBYTE_ORDER._HIGH_LOW , OutVal:=m_maxClosingCurrent );
//			AryByteTo(In:=arrReadData[76] , Size:= 4, Order:=_eBYTE_ORDER._HIGH_LOW , OutVal:=m_readRFIDPos );
	    	iStepRFID:=0;
			iStepRFIDOnLine:=0;
	   ELSE
	        iStepRFID:=30;
	   END_IF
	 30:
	    g_readedRFID:=FALSE;
		GVL_InstruTestUIVars.g_readRFIDFlag:=FALSE;
	    iStepRFID:=0;
		iStepRFIDOnLine:=0;
 	 53:	                   //Write
	  arrReadData:=arrRFIDData;
	  arrSendData:=arrRFIDData;
	  iStepRFID:=55;
     55:  
	  arrSendData[0]:=16#FF;
	  arrSendData[1]:=16#76;  arrSendData[2]:=16#12;
	  arrSendData[3]:=16#00;  arrSendData[4]:=16#01;
	  arrSendData[5]:=16#00;  arrSendData[6]:=16#00;
	  arrSendData[7]:=16#00;  arrSendData[8]:=16#6E;  //Length  //110 BYTE
	  
	//  g_RFIDinstruSN:=g_newInstruSN;
	  //Data
	  arrSendData[11]:=(INT_TO_BYTE(g_moveMode) AND 16#0F) +(INT_TO_BYTE(SHL(g_energyType,4)) AND 16#F0);
	   FOR i:=1 TO 8 BY 1 DO
		  arrSendData[61+i]:=ULINT_TO_BYTE(SHR(g_RFIDinstruSN,64-i*8) );
	  END_FOR
	   FOR i:=1 TO 4 BY 1 DO
		  arrSendData[71+i]:=DINT_TO_BYTE(SHR(m_writeRFIDTimes,32-i*8) );
	  END_FOR
	   FOR i:=1 TO 4 BY 1 DO
		  arrSendData[31+i]:=DINT_TO_BYTE(SHR(LREAL_TO_DINT(m_writeInstrument_pos_L1*1000),32-i*8) );
	  END_FOR
	   FOR i:=1 TO 4 BY 1 DO
		  arrSendData[41+i]:=DINT_TO_BYTE(SHR(LREAL_TO_DINT(m_writeInstrument_pos_L2*1000),32-i*8) );
	  END_FOR
	   FOR i:=1 TO 4 BY 1 DO
		  arrSendData[51+i]:=DINT_TO_BYTE(SHR(LREAL_TO_DINT(m_writeInstrument_pos_L3*1000),32-i*8) );
	  END_FOR
	  
	   uiRFIDWrite:=0;  
	  FOR i:=11 TO 111 BY 1 DO                            //Sum 
		   uiRFIDWrite:=BYTE_TO_UINT(arrSendData[i])+uiRFIDWrite;
	  END_FOR
	  
	  arrSendData[112]:=UINT_TO_BYTE(SHR(uiRFIDWrite,8) );
	  arrSendData[113]:=UINT_TO_BYTE(uiRFIDWrite AND 16#00FF);
                   
	  wCRC16:=MEM.CRC16_Modbus(pMemoryBlock:= ADR(arrSendData ), uiLength:=119 );  //CRC
	  arrSendData[119]:=UINT_TO_BYTE(SHR(wCRC16,8) );
	  arrSendData[120]:=UINT_TO_BYTE(wCRC16 AND 16#00FF);
	  bSend:=TRUE; 
	  iStepRFID:=60;
	60:
	   IF arrReadData[0]<>0  THEN
           iStepRFID:=65;
	   END_IF
	   IF fbTonRFID.Q THEN
	   	   iStepRFID:=0;
		   iStepRFIDOnLine:=0;
	   END_IF
	65: 
	IF fbTonReadData.Q THEN
	   IF arrReadData[5]=0 THEN
	  	   iStepRFID:=75;
	   END_IF
	   IF arrReadData[5]<>0THEN
	   	   iStepRFID:=80;
	   END_IF
	END_IF
	 75:
	   g_writedRFID:=TRUE;
	   iStepRFID:=0;
	   iStepRFIDOnLine:=0;
	 80:
	   g_writedRFID:=FALSE;
	   iStepRFID:=0;
	   iStepRFIDOnLine:=0;
	  
END_CASE
	 (*
SNMid :=LREAL_TO_INT( FLOOR(ULINT_TO_LREAL(uiRFIDReadSN)/1000000000));
g_informationVerificationPassed:=FALSE;
IF g_readedRFID AND g_instruSN=uiRFIDReadSN  AND  (SNMid=042 OR SNMid=043 OR TRUE )AND 
	ABS(GVL_InstruTestUIVars.g_instruZeroPos[1]-m_readInstrument_pos_L1)<0.01 AND
	ABS(GVL_InstruTestUIVars.g_instruZeroPos[2]-m_readInstrument_pos_L2)<0.01 AND
	ABS(GVL_InstruTestUIVars.g_instruZeroPos[3]-m_readInstrument_pos_L3)<0.01 THEN
	
	g_informationVerificationPassed:=TRUE;
END_IF;

*)
IF g_informationVerificationPassed THEN
(*	g_instruPurposeUI:=m_instruPurpose;
	GVL_InstruTestUIVars.g_instruName:=1;
	GVL_InstruTestUIVars.g_numberOfUsableTimesUI:=1;
	GVL_InstruTestUIVars.g_usedTimesUI:=0;
	GVL_InstruTestUIVars.g_maxClosingCurrentUI:=m_maxClosingCurrent;
	IF SNMid=042 THEN
	    GVL_InstruTestUIVars.g_driveRodLengthUI:=464.6;
	    GVL_InstruTestUIVars.g_instruNameEnglish:=1;
		GVL_InstruTestUIVars.g_instruType:=1;
	ELSIF SNMid=043 THEN 
	    GVL_InstruTestUIVars.g_driveRodLengthUI:=552.3;
	    GVL_InstruTestUIVars.g_instruNameEnglish:=2;
		GVL_InstruTestUIVars.g_instruType:=2;
	END_IF
	GVL_InstruTestUIVars.g_maxWorkAngleUI:=45;
	GVL_InstruTestUIVars.g_reductionRatioK1UI:=25;
	GVL_InstruTestUIVars.g_reductionRatioK2UI:=13;
	GVL_InstruTestUIVars.g_reductionRatioK3UI:=18.5;
	GVL_InstruTestUIVars.g_moveModeUI:=5;
	GVL_InstruTestUIVars.g_energyTypeUI:=4;
	GVL_InstruTestUIVars.g_instruVersionUI:=01;
	GVL_InstruTestUIVars.g_formVersionUI:=01;
	GVL_InstruTestUIVars.g_readOpenAngleLinkPos:=DINT_TO_LREAL(m_readPos)/1000;
ELSE 
    GVL_InstruTestUIVars.g_instruPurposeUI:=0;
	GVL_InstruTestUIVars.g_instruName:=0;
	GVL_InstruTestUIVars.g_instruSN:=0;
	GVL_InstruTestUIVars.g_instruType:=0;
	GVL_InstruTestUIVars.g_numberOfUsableTimesUI:=0;
	GVL_InstruTestUIVars.g_usedTimesUI:=0;
	GVL_InstruTestUIVars.g_maxClosingCurrentUI:=0;
	GVL_InstruTestUIVars.g_driveRodLengthUI:=0;
	GVL_InstruTestUIVars.g_maxWorkAngleUI:=0;
	GVL_InstruTestUIVars.g_reductionRatioK1UI:=0;
	GVL_InstruTestUIVars.g_reductionRatioK2UI:=0;
	GVL_InstruTestUIVars.g_reductionRatioK3UI:=0;
	GVL_InstruTestUIVars.g_moveModeUI:=0;
	GVL_InstruTestUIVars.g_energyTypeUI:=0;
	GVL_InstruTestUIVars.g_instruVersionUI:=0;
	GVL_InstruTestUIVars.g_formVersionUI:=0;
	GVL_InstruTestUIVars.g_instruNameEnglish:=0;
	GVL_InstruTestUIVars.g_readOpenAngleLinkPos:=0;
	*)
END_IF
(*
IF m_instrument.onChipData.m_InstruReadSucceed THEN
	GVL_InstruTestUIVars.g_readSNNum:=m_instrument.onChipData.m_InstruseriesNum;
END_IF
GVL_InstruTestUIVars.g_readRFIDFlag:=g_readedRFID;
GVL_InstruTestUIVars.g_offLineRFID:=g_offLineRFID;
GVL_InstruTestUIVars.g_informationVerificationPassed:=g_informationVerificationPassed;
GVL_InstruTestUIVars.g_readedRFID:=g_readedRFID;
GVL_InstruTestUIVars.g_RFID_SN:=ULINT_TO_STRING(uiRFIDReadSN);
IF (LEN(GVL_InstruTestUIVars.g_RFID_SN)=10)THEN
	GVL_InstruTestUIVars.g_RFID_SN:=concat('00',GVL_InstruTestUIVars.g_RFID_SN);
ELSIF  (LEN(GVL_InstruTestUIVars.g_RFID_SN)=11)THEN
	GVL_InstruTestUIVars.g_RFID_SN:=concat('0',GVL_InstruTestUIVars.g_RFID_SN);
ELSE
	GVL_InstruTestUIVars.g_RFID_SN:=GVL_InstruTestUIVars.g_RFID_SN;
END_IF
IF m_instrument.onChipData.m_InstruReadSucceed THEN
	g_instruSN:= GVL_InstruTestUIVars.g_readSNNum;
	g_RFIDinstruSN:=GVL_InstruTestUIVars.g_readSNNum;
	m_writeRFIDTimes:=GVL_InstruTestUIVars.g_instruNumberOfUses;
	m_writeInstrument_pos_L1:=GVL_InstruTestUIVars.g_instruZeroPos[1];
	m_writeInstrument_pos_L2:=GVL_InstruTestUIVars.g_instruZeroPos[2];
	m_writeInstrument_pos_L3:=GVL_InstruTestUIVars.g_instruZeroPos[3];
END_IF
GVL_InstruTestUIVars.m_RFIDTimes:=m_readRFIDTimes;
GVL_InstruTestUIVars.m_Instrument_pos_L1:=m_readInstrument_pos_L1;
GVL_InstruTestUIVars.m_Instrument_pos_L2:=m_readInstrument_pos_L2;
GVL_InstruTestUIVars.m_Instrument_pos_L3:=m_readInstrument_pos_L3;
*)
(*
fbTonRFIDReaded(IN:=(GVL_InstruTestUIVars.IsolationPlate_Instrument_Install_Start AND 16#2)<>16#2,PT:=T#3S);
IF fbTonRFIDReaded.Q THEN
g_readedRFID:=FALSE;
END_IF
*)



//read recipe
IF (m_bReadRecipeStep<=2 AND m_bReadRecipeStep>0) THEN
	//The method loads a recipe from the specified recipe file.  It subsequently writes the recipe into the PLC variables.
    ReturnDwordRead:=RecipeManCommands.LoadAndWriteRecipe(RecipeDefinitionName:=GVL_SystemParameters.RecipeDefinitionName[m_bReadRecipeStep] , RecipeName:='RecipeRecord');
	IF ReturnDwordRead = ERR_OK THEN
		m_bReadRecipeStep:=m_bReadRecipeStep+1; 
	END_IF
END_IF 
//loadConfigFile := m_bReadRecipeStep>2;
//write recipe
IF m_saveAccount THEN	
	//This method creates a new recipe in the specified recipe definition. It subsequently reads the current PLC values into the new recipe and saves it as a recipe file with a standard name.
	 RecipeManCommands.CreateRecipe(RecipeDefinitionName:=GVL_SystemParameters.RecipeDefinitionName[1] , RecipeName:='RecipeRecord' );
	 ReturnDwordWrite:=RecipeManCommands.ReadAndSaveRecipe(RecipeDefinitionName:=GVL_SystemParameters.RecipeDefinitionName[1] , RecipeName:='RecipeRecord' ); 
	 m_saveAccount:=0;
END_IF
IF  m_saveCaliLinkEncoder THEN	
	//This method creates a new recipe in the specified recipe definition. It subsequently reads the current PLC values into the new recipe and saves it as a recipe file with a standard name.
	 RecipeManCommands.CreateRecipe(RecipeDefinitionName:=GVL_SystemParameters.RecipeDefinitionName[2] , RecipeName:='RecipeRecord' );
	 ReturnDwordWrite:=RecipeManCommands.ReadAndSaveRecipe(RecipeDefinitionName:=GVL_SystemParameters.RecipeDefinitionName[2] , RecipeName:='RecipeRecord' );
	 m_saveCaliLinkEncoder:=0;
END_IF

GVL_InstruTestUIVars.g_instruSNLen:=LEN(GVL_InstruTestUIVars.g_newInstruSN);
END_METHOD

METHOD checkLight : BOOL
VAR_INPUT
	i_lightCtrlWord : UDINT;
END_VAR

VAR
	lightCtrlWord : UDINT;
END_VAR
// to PDO
m_lightIO := UDINT_TO_DINT(i_lightCtrlWord);

// trig sdo write
lightCtrlWord := SHL(i_lightCtrlWord,16);
m_SdoWrite[1](sNetId:= m_armNetId, nSlaveAddr:= m_jointAddrJ8, nSubIndex:= 0, nIndex:= 16#6097, pSrcBuf:=ADR(lightCtrlWord) , cbBufLen:=SIZEOF(lightCtrlWord) , bExecute:= TRUE, tTimeout:= , bBusy=> , bError=> , nErrId=> );
m_SdoWrite[2](sNetId:= m_armNetId, nSlaveAddr:= m_jointAddrPbox, nSubIndex:= 0, nIndex:= 16#6097, pSrcBuf:= ADR(lightCtrlWord), cbBufLen:= SIZEOF(lightCtrlWord), bExecute:= TRUE, tTimeout:= , bBusy=> , bError=> , nErrId=> );

// disable sdo write
IF NOT m_SdoWrite[1].bBusy AND  NOT m_SdoWrite[2].bBusy THEN
	m_SdoWrite[1](bExecute:=FALSE);
	m_SdoWrite[2](bExecute:=FALSE);
END_IF
END_METHOD

PROPERTY cmdCartPose : REFERENCE TO ST_Frame
GET
cmdCartPose REF= m_cmdCartPose;
END_GET
END_PROPERTY

PROPERTY cmdCartTwist : REFERENCE to Vec6d
GET
cmdCartTwist REF= m_cmdCartTwist;
END_GET
END_PROPERTY

PROPERTY cmdJntCurrent : REFERENCE TO  Vec8d
GET
cmdJntCurrent ref= m_cmdJntCurrent;
END_GET
END_PROPERTY

PROPERTY cmdJntPos : REFERENCE TO Vec8d
GET
cmdJntPos REF= m_cmdJntPos;
END_GET
END_PROPERTY

PROPERTY cmdJntTrq :REFERENCE TO Vec8d
GET
cmdJntTrq REF= m_cmdJntTrq;
END_GET
END_PROPERTY

PROPERTY cmdJntVel : REFERENCE TO Vec8d
GET
cmdJntVel REF= m_cmdJntVel;
END_GET
END_PROPERTY

PROPERTY curCartPose : REFERENCE TO ST_Frame
GET
curCartPose ref=m_curCartPose;
END_GET
END_PROPERTY

PROPERTY curCartTwist : REFERENCE TO Vec6d
GET
curCartTwist ref=m_curCartTwist;
END_GET
END_PROPERTY

PROPERTY curDHJntPos :REFERENCE TO Vec6d
GET
curDHJntPos ref= m_curDHJntPos;
END_GET
END_PROPERTY

PROPERTY curDHJntVel :REFERENCE TO Vec6d
GET
curDHJntVel REF= m_curDHJntVel;
END_GET
END_PROPERTY

PROPERTY curGripAngle : LREAL
GET
curGripAngle:=m_curGripAngle;
END_GET
END_PROPERTY

PROPERTY curJntPos : REFERENCE TO Vec8d
GET
curJntPos ref=m_curJntPos;
END_GET
END_PROPERTY

PROPERTY curJntTrq : REFERENCE TO Vec8d
GET
curJntTrq ref=m_curJntTrq;
END_GET
END_PROPERTY

PROPERTY curJntVel :REFERENCE TO Vec8d
GET
curJntVel ref=m_curJntVel;
END_GET
END_PROPERTY

PROPERTY curLinkPos :REFERENCE TO Vec8d
GET
curLinkPos ref=m_curLinkPos;
END_GET
END_PROPERTY

PROPERTY curMotorPos : REFERENCE TO  Vec8d
GET
curMotorPos ref=m_curMotorPos;
END_GET
END_PROPERTY

METHOD PUBLIC enable : BOOL
VAR_IN_OUT CONSTANT
	i_jntIdx :Vec8i;
END_VAR
VAR
	i :INT ;
END_VAR
FOR i:=1 TO g_sJntNum DO
	IF 1= i_jntIdx[i] THEN
		m_joints[i].enable();
	ELSE
		m_joints[i].disable();
	END_IF
END_FOR
END_METHOD

PROPERTY filtJntCurrent :REFERENCE TO Vec8d
GET
filtJntCurrent ref= m_filtJntCurrent;
END_GET
END_PROPERTY

// from active joint position to cartesian pose in arm origin
METHOD PROTECTED forwardKinematic : BOOL
VAR_IN_OUT CONSTANT
	i_DHJntPos :Vec6d;
END_VAR
VAR_IN_OUT
	r_cartPose :ST_Frame;
END_VAR
VAR
	d1, L, a, b :LREAL;
	q3 :LREAL;

	c1,c2,c4,c5,c6,c7 :LREAL;
	s1,s2,s4,s5,s6,s7 :LREAL;
	DHRot :Mat3d;
	
	tmpRot1,tmpRot2 : Mat3d;

END_VAR

d1:=GVL_SlaveArmKinematic.g_d1;
L:=m_instrument.instruTypeInfo.m_rodLength;
a:=m_instrument.instruTypeInfo.m_headLength;
b:=m_instrument.instruTypeInfo.m_fingerLength;

q3:=i_DHJntPos[3];
c1:=COS(i_DHJntPos[1]);
c2:=COS(i_DHJntPos[2]);
c4:=COS(i_DHJntPos[4]);
c5:=COS(i_DHJntPos[5]);
c6:=COS(i_DHJntPos[6]);

s1:=SIN(i_DHJntPos[1]);
s2:=SIN(i_DHJntPos[2]);
s4:=SIN(i_DHJntPos[4]);
s5:=SIN(i_DHJntPos[5]);
s6:=SIN(i_DHJntPos[6]);


// cartesian pose frame
r_cartPose.m_pos[1]:=a*(c5*(s1*s4 + c1*c2*c4) - c1*s2*s5) + b*(c6*(c5*(s1*s4 + c1*c2*c4) - c1*s2*s5) - s6*(c4*s1 - c1*c2*s4)) + L*c1*s2 - q3*c1*s2;
r_cartPose.m_pos[2]:=a*(c2*s5 + c4*c5*s2) - d1 - L*c2 + q3*c2 + b*(c6*(c2*s5 + c4*c5*s2) + s2*s4*s6);
r_cartPose.m_pos[3]:=L*s1*s2 - a*(c5*(c1*s4 - c2*c4*s1) + s1*s2*s5) - b*(c6*(c5*(c1*s4 - c2*c4*s1) + s1*s2*s5) - s6*(c1*c4 + c2*s1*s4)) - q3*s1*s2;

DHRot[1,1]:= c6*(c5*(s1*s4 + c1*c2*c4) - c1*s2*s5) - s6*(c4*s1 - c1*c2*s4);
DHRot[2,1]:=c6*(c2*s5 + c4*c5*s2) + s2*s4*s6;
DHRot[3,1]:=s6*(c1*c4 + c2*s1*s4) - c6*(c5*(c1*s4 - c2*c4*s1) + s1*s2*s5);

DHRot[1,2]:=- s6*(c5*(s1*s4 + c1*c2*c4) - c1*s2*s5) - c6*(c4*s1 - c1*c2*s4);
DHRot[2,2]:=c6*s2*s4 - s6*(c2*s5 + c4*c5*s2);
DHRot[3,2]:=s6*(c5*(c1*s4 - c2*c4*s1) + s1*s2*s5) + c6*(c1*c4 + c2*s1*s4);

DHRot[1,3]:= s5*(s1*s4 + c1*c2*c4) + c1*c5*s2;
DHRot[2,3]:= c4*s2*s5 - c2*c5;
DHRot[3,3]:=c5*s1*s2 - s5*(c1*s4 - c2*c4*s1);

// convert to tcp rotation
matMultiply(DHRot, GVL_SlaveArmKinematic.g_tcpRotation, r_cartPOSE.m_rot);

//TODO: need verify
// rotate tcp coordinate 180 degree about z axis if instrument is a head-up 30deg endoscope
IF m_instrument.instruType = InstruType_Endoscope AND m_instrument.curScopeType = EndoScopeType_30 AND m_instrument.curScopePosture = EndoscopePosture_HeadUp THEN
	tmpRot2 := rotZ(pi);
	tmpRot1 := r_cartPOSE.m_rot;
	matMultiply(tmpRot1, tmpRot2, r_cartPOSE.m_rot);
END_IF
END_METHOD

METHOD PUBLIC init : BOOL
VAR_INPUT
	i_armIdx:INT;
END_VAR
VAR 
	i :INT ;
	currentRatioMotor2Jnt: LREAL;
END_VAR
// arm statues init
m_armIdx:=i_armIdx;
m_curGripAngle:=0;
m_simGripAngle:=0;

// joint init
FOR i:=1 TO g_sJntNum DO
	IF i<4 THEN
		m_joints[i].init(m_armIdx, i,g_slaveArmCtrlCycleTime, 1);
	ELSE
		m_joints[i].init(m_armIdx, i,g_slaveArmCtrlCycleTime, 4);
	END_IF
END_FOR

// init joint encoder and position calculation
initJntPos();

// joint controller init
FOR i:=1 TO g_sJntNum DO 
	currentRatioMotor2Jnt:=GVL_SlaveMotorParameters.g_motorTrqConst[i]*GVL_SlaveMotorParameters.g_motorReduction[i]/1000;
	m_jntPIDCtrl[i].init(g_slaveArmCtrlCycleTime,GVL_slaveControlParameters.g_posKp[i],GVL_slaveControlParameters.g_posKd[i],
		GVL_slaveControlParameters.g_posKi[i], GVL_slaveControlParameters.g_posKiLimit[i]* currentRatioMotor2Jnt,
		GVL_slaveControlParameters.g_posCtrlLimit[i]*currentRatioMotor2Jnt);
END_FOR

// instrument init
m_instrument.init(i_armIdx);

//init arm netID and adrr
m_armNetId := GVL_SlaveJointEncoderCaliData.g_slaveArmNetID[armIdx];
m_jointAddrJ8 := GVL_SlaveJointEncoderCaliData.g_slaveJointNetPort[armIdx,3];
m_jointAddrPbox := GVL_SlaveJointEncoderCaliData.g_slaveJointNetPort[armIdx,4];

// endosocpe toggle button check
m_endoscopeTypeSwitch.init(0, 500);
m_endoscopePostureSwitch.init(0,500);
END_METHOD

METHOD PUBLIC initJntPos : BOOL
VAR_INPUT
END_VAR
VAR
	i:INT ;
END_VAR
// joint init
FOR i:=1 TO g_sJntNum DO
	m_joints[i].initJntPos();
END_FOR

// update arm status if joint position is re-init
updateStatus();
END_METHOD

PROPERTY instrument : REFERENCE TO FB_Instrument
GET
instrument REF=m_instrument;
END_GET
END_PROPERTY

PROPERTY instruNear : BOOL
GET
instruNear := m_instruNearFlag;
END_GET
END_PROPERTY

PROPERTY instruOn : bool
GET
instruOn:=m_instruOnFlag;
END_GET
END_PROPERTY

// check if instrument is in ready position(far enough from romote center) for following manipulation
METHOD PUBLIC instruReady : BOOL
VAR_INPUT
END_VAR

VAR
	// check buffer
	checkBuffer :LREAL := 0.005;
END_VAR
IF NOT(m_instrument.onChipData.m_InstruReadSucceed) THEN
	instruReady :=FALSE;
	RETURN;
END_IF

instruReady := m_curJntPos[3] < (m_instrument.instruTypeInfo.m_rodLength+m_instrument.instruTypeInfo.m_headLength
									+ m_instrument.instruTypeInfo.m_fingerLength - GVL_SlaveArmKinematic.g_minInstruRCDis+checkBuffer);
END_METHOD

METHOD PUBLIC isEnabled : BOOL
VAR_IN_OUT CONSTANT
	i_jntIdx :Vec8i;
END_VAR
VAR
	i :INT ;
END_VAR
isEnabled := TRUE;
FOR i:=1 TO g_sJntNum DO
	IF 1= i_jntIdx[i] THEN
		isEnabled :=  (m_joints[i].isEnabled() AND isEnabled);
	END_IF
END_FOR
END_METHOD

PROPERTY isSingurality : bool
GET
isSingurality:=m_isSingularity;
END_GET
END_PROPERTY

PROPERTY jaco :REFERENCE TO Mat6d
GET
jaco ref= m_jaco;
END_GET
END_PROPERTY

PROPERTY jntGravity :REFERENCE TO Vec8d
GET
jntGravity ref=m_jntGravity;
END_GET
END_PROPERTY

PROPERTY linkSingle : REFERENCE TO Vec8d
GET
linkSingle ref=m_curLinkSingle;
END_GET
END_PROPERTY

PROPERTY PUBLIC massMat :REFERENCE TO Mat3d
GET
massMat ref=m_jntMassMat;
END_GET
END_PROPERTY

METHOD mes : BOOL
VAR_INPUT
END_VAR
GVL_MES.g_serialNumLen:=LEN(GVL_MES.g_serialNum);
IF GVL_MES.g_serialNum<>m_serialNumOld AND GVL_MES.g_serialNumLen=9 THEN
	GVL_MES.g_eventTime[1]:=m_time;
END_IF
m_serialNumOld:=GVL_MES.g_serialNum;
GVL_MES.g_actualAccountNumber:=GVL_InstruTestUIVars.g_account.actualAccountNumber;
IF m_logStep=15 THEN
	GVL_MES.g_eventTime[2]:=m_time;
END_IF
GVL_MES.g_powerBoxCalibrationPos:=GVL_SlaveJointEncoderCaliData.g_caliLinkEncoder;
IF GVL_InstruTestUIVars.g_powerBoxCalibrationFlag=FALSE THEN
	GVL_MES.g_eventTime[3]:=m_time;
END_IF
GVL_MES.g_SN:=GVL_InstruTestUIVars.g_instruSN;
IF startFlag THEN
	GVL_MES.g_eventTime[4]:=m_time;
END_IF
GVL_MES.g_writeInstruZeroPos:=GVL_InstruTestUIVars.writeInstruZeroPos;
IF GVL_InstruTestUIVars.g_writeZeroPosFlag THEN
	GVL_MES.g_eventTime[5]:=m_time;
END_IF
GVL_MES.g_instruZeroPos:=GVL_InstruTestUIVars.g_instruZeroPos;
IF startFlag THEN
	GVL_MES.g_eventTime[6]:=m_time;
END_IF
GVL_MES.g_readRFIDFlig:=g_readedRFID;
IF iStepRFID=5 THEN
	GVL_MES.g_eventTime[7]:=m_time;
END_IF
IF GVL_MES.g_autoTestMode=3 OR GVL_MES.g_autoTestMode=13 THEN
	GVL_MES.g_curNumTiredTest:=GVL_InstruTestUIVars.g_curTestCycles;
ELSE
	GVL_MES.g_curNumTiredTest:=0;
END_IF
IF m_curTestCyclesOld<>GVL_InstruTestUIVars.g_curTestCycles AND(GVL_MES.g_autoTestMode=3 OR GVL_MES.g_autoTestMode=13) THEN
	GVL_MES.g_eventTime[8]:=m_time;
END_IF
m_curTestCyclesOld:=GVL_InstruTestUIVars.g_curTestCycles;
IF GVL_MES.g_attitudeOK THEN
	GVL_MES.g_attitudeConfirm:=1;
	GVL_MES.g_attitudeOK:=0;
	GVL_MES.g_eventTime[9]:=m_time;
ELSIF
	GVL_MES.g_attitudeNG THEN
	GVL_MES.g_attitudeConfirm:=2;
	GVL_MES.g_attitudeNG:=0;
	GVL_MES.g_eventTime[9]:=m_time;
END_IF
END_METHOD

METHOD PROTECTED modifyJaco : BOOL
VAR_IN_OUT CONSTANT
	i_DHJntPos :Vec6d;
END_VAR
VAR_IN_OUT
	r_jaco :Mat6d;
END_VAR

VAR CONSTANT
	// modify joint2/3 position to avoid jacobian singularity
	m_Jnt2PosThres :LREAL := -165 * g_deg2Rad;
	m_Jnt3PosThres :LREAL := -0.03;
END_VAR

VAR
	d1, L, a, b :LREAL;
	q2, q3:LREAL;

	c1,c2,c4,c5,c6,c7 :LREAL;
	s1,s2,s4,s5,s6,s7 :LREAL;
END_VAR
d1:=GVL_SlaveArmKinematic.g_d1;
L:=m_instrument.instruTypeInfo.m_rodLength;
a:=m_instrument.instruTypeInfo.m_headLength;
b:=m_instrument.instruTypeInfo.m_fingerLength;

q2 := i_DHJntPos[2];
IF q2 < m_Jnt2PosThres THEN
	q2 := m_Jnt2PosThres;
END_IF

q3:=i_DHJntPos[3];
IF q3 - L > m_Jnt3PosThres THEN
	q3:= L + m_Jnt3PosThres;
END_IF

c1:=COS(i_DHJntPos[1]);
c2:=COS(q2);
c4:=COS(i_DHJntPos[4]);
c5:=COS(i_DHJntPos[5]);
c6:=COS(i_DHJntPos[6]);

s1:=SIN(i_DHJntPos[1]);
s2:=SIN(q2);
s4:=SIN(i_DHJntPos[4]);
s5:=SIN(i_DHJntPos[5]);
s6:=SIN(i_DHJntPos[6]);

// jacobian with DH joints
r_jaco[1,1]:=b*(c6*(c5*(c1*s4 - c2*c4*s1) + s1*s2*s5) - s6*(c1*c4 + c2*s1*s4)) + a*(c5*(c1*s4 - c2*c4*s1) + s1*s2*s5) - L*s1*s2 + q3*s1*s2;
r_jaco[1,2]:=-c1*(a*(c2*s5 + c4*c5*s2) - L*c2 + q3*c2 + b*(c6*(c2*s5 + c4*c5*s2) + s2*s4*s6));
r_jaco[1,3]:=-c1*s2;
r_jaco[1,4]:=s1*s2*(a*(c2*s5 + c4*c5*s2) + b*(c6*(c2*s5 + c4*c5*s2) + s2*s4*s6)) - c2*(b*(c6*(c5*(c1*s4 - c2*c4*s1) + s1*s2*s5) - s6*(c1*c4 + c2*s1*s4)) + a*(c5*(c1*s4 - c2*c4*s1) + s1*s2*s5));
r_jaco[1,5]:=- (a*(c2*s5 + c4*c5*s2) + b*(c6*(c2*s5 + c4*c5*s2) + s2*s4*s6))*(c1*c4 + c2*s1*s4) - s2*s4*(b*(c6*(c5*(c1*s4 - c2*c4*s1) + s1*s2*s5) - s6*(c1*c4 + c2*s1*s4)) + a*(c5*(c1*s4 - c2*c4*s1) + s1*s2*s5));
r_jaco[1,6]:= b*(c6*(c5*(c1*s4 - c2*c4*s1) + s1*s2*s5) - s6*(c1*c4 + c2*s1*s4))*(c2*c5 - c4*s2*s5) + b*(s5*(c1*s4 - c2*c4*s1) - c5*s1*s2)*(c6*(c2*s5 + c4*c5*s2) + s2*s4*s6);


r_jaco[2,1]:=0;
r_jaco[2,2]:=c1*(a*(c5*(s1*s4 + c1*c2*c4) - c1*s2*s5) + b*(c6*(c5*(s1*s4 + c1*c2*c4) - c1*s2*s5) - s6*(c4*s1 - c1*c2*s4)) + L*c1*s2 - q3*c1*s2) - s1*(b*(c6*(c5*(c1*s4 - c2*c4*s1) + s1*s2*s5) - s6*(c1*c4 + c2*s1*s4)) + a*(c5*(c1*s4 - c2*c4*s1) + s1*s2*s5) - L*s1*s2 + q3*s1*s2);
r_jaco[2,3]:= c2;
r_jaco[2,4]:=- s1*s2*(a*(c5*(s1*s4 + c1*c2*c4) - c1*s2*s5) + b*(c6*(c5*(s1*s4 + c1*c2*c4) - c1*s2*s5) - s6*(c4*s1 - c1*c2*s4))) - c1*s2*(b*(c6*(c5*(c1*s4 - c2*c4*s1) + s1*s2*s5) - s6*(c1*c4 + c2*s1*s4)) + a*(c5*(c1*s4 - c2*c4*s1) + s1*s2*s5));
r_jaco[2,5]:=(a*(c5*(s1*s4 + c1*c2*c4) - c1*s2*s5) + b*(c6*(c5*(s1*s4 + c1*c2*c4) - c1*s2*s5) - s6*(c4*s1 - c1*c2*s4)))*(c1*c4 + c2*s1*s4) - (b*(c6*(c5*(c1*s4 - c2*c4*s1) + s1*s2*s5) - s6*(c1*c4 + c2*s1*s4)) + a*(c5*(c1*s4 - c2*c4*s1) + s1*s2*s5))*(c4*s1 - c1*c2*s4);
r_jaco[2,6]:=b*(c6*(c5*(c1*s4 - c2*c4*s1) + s1*s2*s5) - s6*(c1*c4 + c2*s1*s4))*(s5*(s1*s4 + c1*c2*c4) + c1*c5*s2) - b*(s5*(c1*s4 - c2*c4*s1) - c5*s1*s2)*(c6*(c5*(s1*s4 + c1*c2*c4) - c1*s2*s5) - s6*(c4*s1 - c1*c2*s4));

r_jaco[3,1]:=a*(c5*(s1*s4 + c1*c2*c4) - c1*s2*s5) + b*(c6*(c5*(s1*s4 + c1*c2*c4) - c1*s2*s5) - s6*(c4*s1 - c1*c2*s4)) + L*c1*s2 - q3*c1*s2;
r_jaco[3,2]:=-s1*(a*(c2*s5 + c4*c5*s2) - L*c2 + q3*c2 + b*(c6*(c2*s5 + c4*c5*s2) + s2*s4*s6));
r_jaco[3,3]:=-s1*s2;
r_jaco[3,4]:=- c2*(a*(c5*(s1*s4 + c1*c2*c4) - c1*s2*s5) + b*(c6*(c5*(s1*s4 + c1*c2*c4) - c1*s2*s5) - s6*(c4*s1 - c1*c2*s4))) - c1*s2*(a*(c2*s5 + c4*c5*s2) + b*(c6*(c2*s5 + c4*c5*s2) + s2*s4*s6));
r_jaco[3,5]:=- (a*(c2*s5 + c4*c5*s2) + b*(c6*(c2*s5 + c4*c5*s2) + s2*s4*s6))*(c4*s1 - c1*c2*s4) - s2*s4*(a*(c5*(s1*s4 + c1*c2*c4) - c1*s2*s5) + b*(c6*(c5*(s1*s4 + c1*c2*c4) - c1*s2*s5) - s6*(c4*s1 - c1*c2*s4)));
r_jaco[3,6]:=b*(c6*(c5*(s1*s4 + c1*c2*c4) - c1*s2*s5) - s6*(c4*s1 - c1*c2*s4))*(c2*c5 - c4*s2*s5) + b*(c6*(c2*s5 + c4*c5*s2) + s2*s4*s6)*(s5*(s1*s4 + c1*c2*c4) + c1*c5*s2);

r_jaco[4,1]:=0;
r_jaco[4,2]:=-s1;
r_jaco[4,3]:=0;
r_jaco[4,4]:=-c1*s2;
r_jaco[4,5]:=c1*c2*s4 - c4*s1;
r_jaco[4,6]:=s5*(s1*s4 + c1*c2*c4) + c1*c5*s2;

r_jaco[5,1]:=-1;
r_jaco[5,2]:=0;
r_jaco[5,3]:=0;
r_jaco[5,4]:=c2;
r_jaco[5,5]:=s2*s4;
r_jaco[5,6]:=c4*s2*s5 - c2*c5;

r_jaco[6,1]:=0;
r_jaco[6,2]:=c1;
r_jaco[6,3]:=0;
r_jaco[6,4]:=-s1*s2;
r_jaco[6,5]:=c1*c4 + c2*s1*s4;
r_jaco[6,6]:=c5*s1*s2 - s5*(c1*s4 - c2*c4*s1);
END_METHOD

PROPERTY panelOn : bool
GET
panelOn :=m_panelOnFlag;
END_GET
END_PROPERTY

PROPERTY rawJntCurrent :REFERENCE TO Vec8d
GET
rawJntCurrent ref=m_rawJntCurrent;
END_GET
END_PROPERTY

// check if instrument is in ready position(far enough from romote center) for following manipulation
METHOD PUBLIC readyForInstruMount : BOOL
VAR_INPUT
END_VAR

VAR
	// check buffer
	checkBuffer :LREAL := 0.01;
END_VAR
readyForInstruMount := (m_curJntPos[3]> GVL_SlaveMotorParameters.g_maxDHJntPos[3]-checkBuffer AND m_panelOnFlag);
END_METHOD

METHOD PUBLIC resetInstruDepth : BOOL
VAR_INPUT
END_VAR
m_instruInvasionDepth :=GVL_SlaveMotorParameters.g_maxJntPos[3];
END_METHOD

METHOD PUBLIC setInstruDepth : BOOL
VAR_INPUT
END_VAR
m_instruInvasionDepth := m_curJntPos[3]-m_instrument.instruTypeInfo.m_rodLength-m_instrument.instruTypeInfo.m_headLength
						- m_instrument.instruTypeInfo.m_fingerLength;
END_METHOD

METHOD setSaveCaliLinkEncoder : BOOL
VAR_INPUT
END_VAR
m_saveCaliLinkEncoder:=1;
END_METHOD

PROPERTY simCartPose :REFERENCE TO ST_Frame
GET
simCartPose ref=m_simCartPose;
END_GET
END_PROPERTY

PROPERTY simDHJntPos :REFERENCE TO Vec6d
GET
simDHJntPos ref= m_simDHJntPos;
END_GET
END_PROPERTY

PROPERTY simGripAngle : LREAL
GET
simGripAngle:=m_simGripAngle;
END_GET
END_PROPERTY

PROPERTY simJaco :REFERENCE TO mat6d
GET
simJaco ref=m_simJaco;
END_GET
END_PROPERTY

PROPERTY simJacoInv :REFERENCE TO Mat6d
GET
simJacoInv ref= m_simJacoInv;
END_GET
END_PROPERTY

PROPERTY PUBLIC trocarOn : bool
GET
trocarOn := m_trocarOnFlag;
END_GET
END_PROPERTY

// update joints control command
METHOD PUBLIC updateCmds : BOOL
VAR_IN_OUT CONSTANT
	i_armCtrlCmd : ST_SlaveArmCtrlCmds;
END_VAR
VAR
	i:INT;
END_VAR
m_cmdJntTrq:=i_armCtrlCmd.m_cmdJntTrq;
m_cmdJntPos :=i_armCtrlCmd.m_cmdJntPos;
m_cmdJntVel :=i_armCtrlCmd.m_cmdJntVel;
m_cmdCartTwist := i_armCtrlCmd.m_cmdCartTwist;
m_cmdCartPose :=i_armCtrlCmd.m_cmdCartPose;
m_simJntPos:=i_armCtrlCmd.m_simJntPos;

// update simulated master arm
updateSimStatus();

// enable/disable joints
enable(i_armCtrlCmd.m_jntEnableFlag);

m_codeTime(START:=TRUE, RESET:=TRUE);
// position/torque control
FOR i:=1 TO g_sJntNum DO 
	m_joints[i].setMaxCurrent(GVL_InstruTestUIVars.g_actualRatedCurrent[i]);
	IF i_armCtrlCmd.m_jntOPMode[i]=DriverOPMode_PosTrq THEN
		// position controller and gravity feedforward
		m_cmdJntTrq[i]:=m_jntPIDCtrl[i].run(m_cmdJntPos[i],m_curJntPos[i],m_cmdJntVel[i],m_curJntVel[i]);
		m_cmdJntTrq[i]:=m_cmdJntTrq[i]+m_jntGravity[i] + i_armCtrlCmd.m_FFJntTrq[i];
		m_joints[i].updateCmds(DriverOPMode_Trq,m_cmdJntPos[i],m_cmdJntTrq[i]);
	ELSIF i_armCtrlCmd.m_jntOPMode[i]=DriverOPMode_Trq THEN
		// gravity feedforward
		m_jntPIDCtrl[i].reset();
		m_cmdJntTrq[i]:=m_cmdJntTrq[i]+m_jntGravity[i];
		m_joints[i].updateCmds(DriverOPMode_Trq,m_cmdJntPos[i],m_cmdJntTrq[i]);
	ELSE
		m_jntPIDCtrl[i].reset();
		m_cmdJntTrq[i]:=0;
		m_joints[i].updateCmds(DriverOPMode_Pos,m_cmdJntPos[i],m_cmdJntTrq[i]);
	END_IF
	
END_FOR
m_codeTime(START:=FALSE);
END_METHOD

METHOD PUBLIC updateDyna : BOOL
VAR_IN_out constant
	slaveDynaData : ST_SlaveDynaData;
END_VAR
m_jntMassMat:=slaveDynaData.m_massMat[m_armIdx];
m_jntGravity[1]:=slaveDynaData.m_gravity[m_armIdx][1];
m_jntGravity[2]:=slaveDynaData.m_gravity[m_armIdx][2];
m_jntGravity[3]:=slaveDynaData.m_gravity[m_armIdx][3];
END_METHOD

METHOD PUBLIC updateSimStatus : BOOL
VAR_INPUT
END_VAR
//IF m_instrument.ready THEN
	// instrument kinematic
	m_instrument.instruFK(m_simJntPos, m_simDHJntPos, m_simGripAngle);

	// simulated cartesion pose 
	forwardKinematic(m_simDHJntPos,m_simCartPose);
	
	// simulated jacobian
	modifyJaco(m_simDHJntPos,m_simJaco);
	m_isSingularity:=NOT(invMat6(m_simJaco, m_simJacoInv));
//END_IF
END_METHOD

// update arm status, including kinematic and dynamic
METHOD PUBLIC updateStatus : BOOL
VAR_INPUT
END_VAR
VAR 
	i,j:INT;
END_VAR
// update joint data
FOR i:=1 TO g_sJntNum DO
	m_joints[i].updateStatus();
END_FOR

// check IO informantion
checkIO();

//mes
mes();

// get joint data
FOR i:=1 TO g_sJntNum DO
	m_curMotorPos[i]:=m_joints[i].motorPos;
	m_curLinkPos[i]:=m_joints[i].linkPos;
	m_curLinkSingle[i]:=m_joints[i].linkSingle;
	m_curJntPos[i]:=m_joints[i].jntPos;
	m_curJntVel[i]:=m_joints[i].jntVel;
	m_curJntTrq[i]:=m_joints[i].jntTrq;
	m_rawJntCurrent[i]:=m_joints[i].rawCurrent;
	m_filtJntCurrent[i]:=m_joints[i].filtCurrent;
	m_cmdJntCurrent[i]:=m_joints[i].cmdCurrent;
END_FOR 

// only update carteisn data when instrument is ready
//IF m_instrument.ready THEN
	
	// instrument kinematic
	m_instrument.instruFK(m_curJntPos, m_curDHJntPos, m_curGripAngle);

	// cartesion pose
	forwardKinematic(m_curDHJntPos,m_curCartPose);
	
	// jacobian
	calcJaco(m_curDHJntPos,m_jaco);
	
	// DH joint velocity
	m_instrument.instruJntVelFK(m_curJntVel, m_curDHJntVel);
	
	// cartesian twist
	matMultiVec(m_jaco, m_curDHJntVel, m_curCartTwist);
//END_IF
END_METHOD

END_FUNCTION_BLOCK

(* stored: Version 1.1.0.1, ProductVersion 3.1.4024.11
   POU FB_SlaveArm: Id {623926f8-06e2-46b6-bb1f-baa6bc16e9cb}, SpecialFunc None
   Folder property: Id {4aa1799c-1556-4bc1-a713-06f14faa00f1}
   Property adjustFallEdge: Id {892fbc5d-bccd-475a-836d-3ab99edcd203}
   Get Get: Id {e41aaa50-cc49-4924-aa5c-7939e5c2aefd}
   Property adjustOn: Id {afc98598-ed29-4176-9f45-d842c4ec164a}
   Get Get: Id {d84a6e3e-5b0e-406e-b7c3-ff6a74a84739}
   Property armIdx: Id {1bcadfc3-0a4f-4bee-a1a7-b6d4d3a1eb58}
   Get Get: Id {198387ec-2e24-42e6-b0c2-2f769705d46f}
   Method calcJaco: Id {1172e5e4-b7f2-4690-a821-6304414cea84}
   Method checkIO: Id {613633aa-f5bc-4224-95e6-e974a90f8e6a}
   Method checkLight: Id {f01081ee-1e3d-4082-9296-257b5773b0af}
   Property cmdCartPose: Id {72bf034f-e694-478b-8fc6-77f6ebb37ccd}
   Get Get: Id {cf508e47-c40b-4af1-9748-e64ccbaeea52}
   Property cmdCartTwist: Id {db564f7b-db8f-4a3a-ba4b-526788bb30bd}
   Get Get: Id {8a565392-e659-4e2f-8d16-f053ffd74289}
   Property cmdJntCurrent: Id {cbd7aa84-e545-47b8-bdc5-960aa8409c91}
   Get Get: Id {12be56c2-8b79-47d6-b1f2-86b8e0a5f91a}
   Property cmdJntPos: Id {fe3eaf75-296c-46e0-a9c6-f78064c649e8}
   Get Get: Id {21440cc7-9bce-4ec3-adb3-863b046ec9da}
   Property cmdJntTrq: Id {a8b8f509-6313-4dea-add6-0d9f63644d17}
   Get Get: Id {69ae4f04-ab57-4161-852a-de73ff986ad6}
   Property cmdJntVel: Id {8b50ea35-c0ee-4521-ab63-6cd2fbfd419a}
   Get Get: Id {32d77105-7aae-4d69-88ee-4b488832fd1d}
   Property curCartPose: Id {d18be23c-99e5-435e-8688-90e0fb3be9ca}
   Get Get: Id {013b03f6-adb7-4855-b0fe-353f77f67094}
   Property curCartTwist: Id {e4b7010c-887c-41fa-8766-1a9192e9d06a}
   Get Get: Id {b7c89bf7-90fc-4841-be25-e467b1918b68}
   Property curDHJntPos: Id {a2be2c30-01e0-4901-99e6-385cb59adf34}
   Get Get: Id {5292b7b6-7cd6-4d1f-a863-39df8105a863}
   Property curDHJntVel: Id {e70b9eba-b60c-47ce-ba40-0d867f7d1681}
   Get Get: Id {f89a1342-80b1-4a57-8483-5c3af208683c}
   Property curGripAngle: Id {5187a911-df75-4b56-8b45-38142d9b24de}
   Get Get: Id {871729fd-1ba1-4906-aec3-7d572491feb2}
   Property curJntPos: Id {d72c054a-bae9-44cb-97ff-fe7c76c53cb8}
   Get Get: Id {332d5297-fb56-44bd-a751-714464e0813c}
   Property curJntTrq: Id {8c78ba58-302c-4844-9d36-e487700a0e19}
   Get Get: Id {1767bffb-cddd-4133-ad6f-5125f86340af}
   Property curJntVel: Id {904c68d5-30c9-4ed3-b3c5-6bcd345bcd5a}
   Get Get: Id {0a508621-c577-4d50-8cc3-bd8133f79f72}
   Property curLinkPos: Id {3725bf51-2c50-4574-b2a7-e2af9fd4da29}
   Get Get: Id {cff7c92f-5276-4a58-b7ca-f6248868b409}
   Property curMotorPos: Id {ad9d9e24-10f4-4dc4-b0d2-86517dead53b}
   Get Get: Id {bc557e46-3cdd-47ba-9e7f-cf7525f3969d}
   Method enable: Id {596f2892-08b6-4851-84d5-1537c558264e}
   Property filtJntCurrent: Id {1f5e4c97-ef8c-417a-90ec-656c048c0e4f}
   Get Get: Id {34ea0c3d-b0bc-4adb-bbb3-f4ab6640a7ff}
   Method forwardKinematic: Id {182b544f-f7c4-475e-8af7-8c07aa230234}
   Method init: Id {d7bcc040-c32e-4455-ab43-70de0dc2919e}
   Method initJntPos: Id {56ee4071-fcb1-4318-b1b9-837ea21e1627}
   Property instrument: Id {ef5d0758-d499-4e04-a177-87950f9a716b}
   Get Get: Id {3a5249de-ec45-4e88-a302-3df6650a3ff5}
   Property instruNear: Id {29bf66f9-822d-4749-92c9-ee092b53b459}
   Get Get: Id {6b30ea9b-f7b2-4aff-9934-1c8f2b6bc1de}
   Property instruOn: Id {4486d0c9-79b0-4e6c-acfb-23ca16ba44f5}
   Get Get: Id {daa69233-49df-439c-8476-605873205ebf}
   Method instruReady: Id {4f7fb741-1810-447d-a3ef-fca916ec7903}
   Method isEnabled: Id {00a67cf8-62b1-4004-a2ca-9469bb0f3cab}
   Property isSingurality: Id {da3c3ca8-d645-443c-af9d-86ff4ca01cff}
   Get Get: Id {69dc0611-36d4-4919-91ba-cfdefe53366b}
   Property jaco: Id {2c2ce445-b511-4254-9c8e-e5667e1b6bdb}
   Get Get: Id {27a6e900-c6e6-40c0-aa03-4dc0d1214554}
   Property jntGravity: Id {72dbb3a4-f37f-4edd-afb1-2190cd1f62fc}
   Get Get: Id {5c8a2ae5-eaad-400d-b638-ec46a75b5ccb}
   Property linkSingle: Id {23452807-9686-4e19-a62d-225c05ba29f3}
   Get Get: Id {f3f0fe9c-39ae-4e13-ac6a-e473233979ba}
   Property massMat: Id {c4fbf6a1-1d71-4f80-9bfa-395c19261a6f}
   Get Get: Id {b8079ba8-3835-474b-9d8e-6afd86dc6a9b}
   Method mes: Id {76588c5b-a490-47ba-bff5-2070f32dad84}
   Method modifyJaco: Id {d0ec41d7-ce80-43b2-a117-9fcbd2b4368b}
   Property panelOn: Id {38ffa1da-012d-4dbc-ad5b-314577ed285b}
   Get Get: Id {b8c5f533-4196-44c4-9a48-01cc1ca3c250}
   Property rawJntCurrent: Id {f1221838-7bcd-4d84-b9f8-7dc96a864978}
   Get Get: Id {23a8503d-4e33-47db-b530-039bdd0d530f}
   Method readyForInstruMount: Id {70a1cabf-0568-4973-adb8-2d2bf84e7996}
   Method resetInstruDepth: Id {442cf664-eb0b-4d84-a453-ceda2815dd97}
   Method setInstruDepth: Id {f666f43c-697b-4bc4-8326-000cbf8a2e4d}
   Method setSaveCaliLinkEncoder: Id {b8308202-10fd-4610-ad6f-7e31e2afd5e3}
   Property simCartPose: Id {6426ffc4-f74f-4984-ac32-a9f9d8b8c8ca}
   Get Get: Id {a61bb7de-a7ad-4b34-8063-e53c825d0db4}
   Property simDHJntPos: Id {c6c26215-f204-4db3-9793-ef759045910e}
   Get Get: Id {52d60fe7-649d-4c54-a901-14c6c6eee89d}
   Property simGripAngle: Id {4ec8904f-ef0e-46d6-9b7d-280a45e21cf5}
   Get Get: Id {6dc37561-5d97-45fe-bee2-ebd740ec58ce}
   Property simJaco: Id {0fa24ffb-bfb3-496c-82de-08842f53e6e4}
   Get Get: Id {35c7dda2-112e-4042-99cd-4eac5d67ff5e}
   Property simJacoInv: Id {9bccb200-445a-4f96-a4eb-1e257b2cb058}
   Get Get: Id {2b6988d5-cc9a-4745-b2b4-b07fc10b1b71}
   Property trocarOn: Id {ad96c106-befc-48a9-abe7-5d7b42881f88}
   Get Get: Id {bb55ac1e-1079-48fa-ba1e-bc9844803f5a}
   Method updateCmds: Id {4f271d3a-4b2b-4f85-986e-f8fdffb5994c}
   Method updateDyna: Id {02de28e3-c8a7-46cf-834a-5bf048b5e039}
   Method updateSimStatus: Id {f15ad7c2-6655-4b50-9555-9aa968e8753f}
   Method updateStatus: Id {21b3fe9a-0eba-4313-bb9a-33b1f0038771} *)
